// TIA Portal project "SW-Ixxx-xxxx-01" (V15.1)
// Pruebas

(* hardware
DEVICE "S7-1200 station_1"  S7-1200 Station
   slot 0: "Rack_0"  S7-1200 Rack  Rack  V1.0
   slot 1: "PLC_1"  CPU 1211C DC/DC/Rly  6ES7 211-1HE40-0XB0  V4.2
DEVICE "HMI_1"  KTP400 Basic PN
   slot 0: "HMI_1"  KTP400 Basic PN  6AV2 123-2DB03-0AX0  15.1.0.0
   slot 1: "HMI_RT_1"  KTP400 Basic PN  6AV2 123-2DB03-0AX0  15.1.0.0
   slot 5: "HMI_1.IE_CP_1"  PROFINET Interface  15.0.1.0
      slot 1: "Interfaz PROFINET_1"  PROFINET Interface
         slot 1: "Port_1"  Port
*)

// ===== PLC "PLC_1"  CPU 1211C DC/DC/Rly =====

VAR_GLOBAL   // PLC tag table "Tabla de variables estándar"
   "Clock_Byte" AT %MB0 : Byte;
   "Clock_10Hz" AT %M0.0 : Bool;
   "Clock_5Hz" AT %M0.1 : Bool;
   "Clock_2.5Hz" AT %M0.2 : Bool;
   "Clock_2Hz" AT %M0.3 : Bool;
   "Clock_1.25Hz" AT %M0.4 : Bool;
   "Clock_1Hz" AT %M0.5 : Bool;
   "Clock_0.625Hz" AT %M0.6 : Bool;
   "Clock_0.5Hz" AT %M0.7 : Bool;
   "System_Byte" AT %MB1 : Byte;
   "FirstScan" AT %M1.0 : Bool;
   "DiagStatusUpdate" AT %M1.1 : Bool;
   "AlwaysTRUE" AT %M1.2 : Bool;
   "AlwaysFALSE" AT %M1.3 : Bool;
   "Siempre0_IT" AT %M2.0 : Bool;
   "Siempre1_IT" AT %M2.1 : Bool;
   "Debug_IT" AT %M2.2 : Bool;
END_VAR

TYPE "UDT_Motores"
   STRUCT
      Local : Bool;
      Remoto : Bool;
      Manual : Bool;
      Automatico : Bool;
      Habilitado : Bool;
      Deshabilitado : Bool;
      Motor_Ready : Bool;
      Marcha : Bool;
      Confirmacion_de_marcha : Bool;
      Parada : Bool;
      Reset_segundero : Bool;
      Reset_horometro : Bool;
      Comm_PLC_VDF : Bool;   // 1 = OK; 0 = Sin comunicación
      ReservaBool_6 : Bool;
      ReservaBool_7 : Bool;
      ReservaBool_8 : Bool;   // 1= con al menos un enclavamiento activo
      Segundero : Real;   // Segundos en funcionamiento
      Horometro : Real;   // Horas en funcionamiento
      Estado : Real;   // 0 = s/Alm, 1 = c/AlmACK, 2 = c/AlmNoACK, 3 = CondicInseg
      Enclavamiento : Array[0..15] of Bool;
      Alarma : Array[0..15] of Bool;
      VDF : "UDT_VDF";
   END_STRUCT;
   // // Alarma[0] : Falla arranque
   // // Alarma[1] : Falla parada
   // // Alarma[2] : Falla interruptor
   // // Alarma[3] : Falla VDF
   // // Enclavamiento[0] : Equipo enclavado
   // // Enclavamiento[2] : Enclavamiento 2
   // // Enclavamiento[1] : Enclavamiento 1
   // // Enclavamiento[3] : Enclavamiento 3
   // // Enclavamiento[4] : Enclavamiento 4
   // // Enclavamiento[5] : Enclavamiento 5
   // // Enclavamiento[6] : Enclavamiento 6
   // // Enclavamiento[7] : Enclavamiento 7
   // // Enclavamiento[8] : Enclavamiento 8
   // // Enclavamiento[9] : Enclavamiento 9
   // // Enclavamiento[10] : Enclavamiento 10
   // // Enclavamiento[11] : Enclavamiento 11
   // // Enclavamiento[12] : Enclavamiento 12
   // // Enclavamiento[13] : Enclavamiento 13
   // // Enclavamiento[14] : Enclavamiento 14
   // // Enclavamiento[15] : Enclavamiento 15
END_TYPE

TYPE "UDT_Valvulas"
   STRUCT
      Local : Bool;
      Remoto : Bool;
      Manual : Bool;
      Automatico : Bool;
      Habilitado : Bool;
      Deshabilitado : Bool;
      Apertura : Bool;
      Confirmacion_de_apertura : Bool;
      Cierre : Bool;
      Reset_segundero : Bool;
      Reset_horometro : Bool;
      Abriendo : Bool;
      Cerrando : Bool;
      ReservaBool_13 : Bool;
      ReservaBool_14 : Bool;
      ReservaBool_15 : Bool;
      Segundero : Real;   // Segundos en funcionamiento
      Horometro : Real;   // Horas en funcionamiento
      Estado : Real;   // 0 = s/Alm, 1 = c/AlmACK, 2 = c/AlmNoACK, 3 = CondicInseg
      Enclavamiento : Array[0..15] of Bool;
      Alarma : Array[0..15] of Bool;
   END_STRUCT;
   // // Alarma[0] : Falla apertura
   // // Alarma[1] : Falla cierre
   // // Enclavamiento[0] : Equipo enclavado
   // // Enclavamiento[1] : Enclavamiento 1
   // // Enclavamiento[2] : Enclavamiento 2
   // // Enclavamiento[3] : Enclavamiento 3
   // // Enclavamiento[4] : Enclavamiento 4
   // // Enclavamiento[5] : Enclavamiento 5
   // // Enclavamiento[6] : Enclavamiento 6
   // // Enclavamiento[7] : Enclavamiento 7
   // // Enclavamiento[8] : Enclavamiento 8
   // // Enclavamiento[9] : Enclavamiento 9
   // // Enclavamiento[10] : Enclavamiento 10
   // // Enclavamiento[11] : Enclavamiento 11
   // // Enclavamiento[12] : Enclavamiento 12
   // // Enclavamiento[13] : Enclavamiento 13
   // // Enclavamiento[14] : Enclavamiento 14
   // // Enclavamiento[15] : Enclavamiento 15
END_TYPE

TYPE "UDT_Instrumentos"
   STRUCT
      Habilitacion_forzado : Bool;
      Forzado : Bool;
      Reconocer_alarmas_HMI : Bool;
      Reset_valor_acumulado_HMI : Bool;
      Reserva_3 : Bool;
      Reserva_4 : Bool;
      Reserva_5 : Bool;
      Reserva_6 : Bool;
      Reserva_7 : Bool;
      Reserva_8 : Bool;
      Reserva_9 : Bool;
      Reserva_10 : Bool;
      Reserva_11 : Bool;
      Reserva_12 : Bool;
      Reserva_13 : Bool;
      Reserva_14 : Bool;
      Valor_medido : Int;
      Valor_normalizado : Real;
      Valor_escalado : Real;
      Valor_escalado_x_seg : Real;
      Valor_acumulado : Real;
      Seteo : Array[0..6] of Real;
      Alarma : Array[0..15] of Bool;
   END_STRUCT;
   // // Alarma[0] : Alarma por Valor HH
   // // Alarma[1] : Alarma por Valor H
   // // Alarma[2] : Alarma por Valor L
   // // Alarma[3] : Alarma por Valor LL
   // // Alarma[4] : Fuera de Rango
   // // Seteo[0] : Valor de Forzado
   // // Seteo[1] : Valor escalado superior
   // // Seteo[2] : Valor escalado inferior
   // // Seteo[3] : Valor Alarma HH
   // // Seteo[4] : Valor Alarma H
   // // Seteo[5] : Valor Alarma L
   // // Seteo[6] : Valor Alarma LL
END_TYPE

TYPE "UDT_Generadores"
   STRUCT
      Local : Bool;
      Remoto : Bool;
      Manual : Bool;
      Automatico : Bool;
      Habilitado : Bool;
      Deshabilitado : Bool;
      Marcha : Bool;   // Comando marcha/arranque GE
      Confirmacion_de_marcha : Bool;   // 1 = En marcha; 0 = Detenido
      Parada : Bool;   // Comando parada/apagado GE
      Rearranque_automatico : Bool;   // ReEnvío automático del comando marcha/arranque GE
      Reset_horometro : Bool;
      Comm_PLC_GE : Bool;   // 1 = OK; 0 = Sin comunicación
      Ready : Bool;
      Listo_para_carga : Bool;
      En_calentamiento : Bool;   // Inicio espera calentamiento GE
      Confirmacion_calentamiento : Bool;   // Calentamiento Generador OK
      Estado_Generador : Int;   // 0 = Apagado; 1 = En arranque; 2 = Listo para Carga; 3 = En Calentamiento
      Cant_arranques_falla : Int;
      Cant_max_rearranques : Int;
      Calentamiento_et_seg : Int;
      Tiempo_apagado_et_Seg : Int;
      Tiempo_calentamiento : Time;
      Segundero : Real;   // Segundos en funcionamiento
      Horometro : Real;   // Horas en funcionamiento
      Estado : Real;   // 0 = s/Alm, 1 = c/AlmACK, 2 = c/AlmNoACK, 3 = CondicInseg
      Enclavamiento : Array[0..15] of Bool;
      Alarma : Array[0..15] of Bool;
   END_STRUCT;
   // // Alarma[0] : Falla al arrancar GE
   // // Alarma[1] : Falla al detenerse GE
   // // Alarma[2] : Alerta de combustible bajo GE
   // // Alarma[3] : Alarma General
   // // Alarma[4] : Falla comunicación con PLC
   // // Enclavamiento[0] : Equipo enclavado
   // // Enclavamiento[1] : Enclavamiento 1
   // // Enclavamiento[2] : Enclavamiento 2
   // // Enclavamiento[3] : Enclavamiento 3
   // // Enclavamiento[4] : Enclavamiento 4
   // // Enclavamiento[5] : Enclavamiento 5
   // // Enclavamiento[6] : Enclavamiento 6
   // // Enclavamiento[7] : Enclavamiento 7
   // // Enclavamiento[8] : Enclavamiento 8
   // // Enclavamiento[9] : Enclavamiento 9
   // // Enclavamiento[10] : Enclavamiento 10
   // // Enclavamiento[11] : Enclavamiento 11
   // // Enclavamiento[12] : Enclavamiento 12
   // // Enclavamiento[13] : Enclavamiento 13
   // // Enclavamiento[14] : Enclavamiento 14
   // // Enclavamiento[15] : Enclavamiento 15
END_TYPE

TYPE "UDT_VDF"
   STRUCT
      Velocidad_RPM_ref : Real;
      Intensidad_ref : Real;
      Tension_ref : Real;
      Potencia_ref : Real;
      Ret_val : Int;
      Telegrama_Control : Array[0..15] of Word;
      Telegrama_Estado : Array[0..15] of Word;
   END_STRUCT;
   // // Telegrama_Control[0] : Palabra de mando 1 (STW1)
   // // Telegrama_Control[1] : Consigna principal de velocidad
   // // Telegrama_Estado[0] : Palabra de estado 1 (ZSW1)
   // // Telegrama_Estado[1] : Intensidad real Valor absoluto filtrado
   // // Telegrama_Estado[2] : Tensión de salida filtrada
   // // Telegrama_Estado[3] : Velocidad real filtrada
   // // Telegrama_Estado[4] : Potencia activa real filtrada
   // // Telegrama_Estado[5] : Temperatura en motor
   // // Telegrama_Estado[6] : Frecuencia de salida
   // // Telegrama_Estado[7] : Intensidad de fase Valor real, Suma U, V, W
   // // Telegrama_Estado[8] : Código de fallo actual (FAULT_CODE)
   // // Telegrama_Estado[9] : CU Entradas digitales Estado
   // // Telegrama_Estado[10] : Palabra de estado 2
   // // Telegrama_Estado[11] : Tensión en circuito intermedio Valor real
END_TYPE

// folder: B_FUNCIONES GENERALES/DBs Funciones Generales

DATA_BLOCK "DB_Entradas"   // DB100
{ S7_Optimized_Access := 'FALSE' }
VERSION : 0.1
BEGIN
END_DATA_BLOCK

DATA_BLOCK "DB_Salidas"   // DB101
{ S7_Optimized_Access := 'FALSE' }
VERSION : 0.1
BEGIN
END_DATA_BLOCK

DATA_BLOCK "DB_Enclavamientos"   // DB110
{ S7_Optimized_Access := 'FALSE' }
VERSION : 0.1
BEGIN
END_DATA_BLOCK

DATA_BLOCK "DB_PIDs"   // DB120
{ S7_Optimized_Access := 'FALSE' }
VERSION : 0.1
BEGIN
END_DATA_BLOCK

// folder: C_MOTORES/DBs Motores

DATA_BLOCK "DB_Bombas"   // DB210
{ S7_Optimized_Access := 'FALSE' }
VERSION : 0.1
   VAR
      Bomba1 : "UDT_Motores";
   END_VAR
BEGIN
END_DATA_BLOCK

DATA_BLOCK "DB_Agitadores"   // DB220
{ S7_Optimized_Access := 'FALSE' }
VERSION : 0.1
   VAR
      Agitador1 : "UDT_Motores";
   END_VAR
BEGIN
END_DATA_BLOCK

DATA_BLOCK "DB_Ventiladores"   // DB230
{ S7_Optimized_Access := 'FALSE' }
VERSION : 0.1
   VAR
      Ventilador1 : "UDT_Motores";
   END_VAR
BEGIN
END_DATA_BLOCK

DATA_BLOCK "DB_Cintas"   // DB240
{ S7_Optimized_Access := 'FALSE' }
VERSION : 0.1
   VAR
      Cinta1 : "UDT_Motores";
   END_VAR
BEGIN
END_DATA_BLOCK

// folder: D_VALVULAS/DBs Válvulas

DATA_BLOCK "DB_Valvulas_Solenoides"   // DB310
{ S7_Optimized_Access := 'FALSE' }
VERSION : 0.1
BEGIN
END_DATA_BLOCK

DATA_BLOCK "BLQ_Valvula_Solenoide_0_DB"   // DB311
{ S7_Optimized_Access := 'FALSE' }
VERSION : 0.1
// stored: InstanceOfName BLQ_Valvula_Solenoide
"BLQ_Valvula_Solenoide"
BEGIN
END_DATA_BLOCK

DATA_BLOCK "DB_Valvulas_de_Control"   // DB320
{ S7_Optimized_Access := 'FALSE' }
VERSION : 0.1
BEGIN
END_DATA_BLOCK

// folder: E_INSTRUMENTOS/DBs Instrumentos

DATA_BLOCK "DB_Caudalimetros"   // DB410
{ S7_Optimized_Access := 'FALSE' }
VERSION : 0.1
   VAR
      FIT1 : "UDT_Instrumentos";
   END_VAR
BEGIN
END_DATA_BLOCK

DATA_BLOCK "BLQ_FIT_0_DB"   // DB411
{ S7_Optimized_Access := 'FALSE' }
VERSION : 0.1
// stored: InstanceOfName BLQ_Inst_Analogico
"BLQ_Inst_Analogico"
BEGIN
END_DATA_BLOCK

DATA_BLOCK "DB_Sensores_Nivel"   // DB420
{ S7_Optimized_Access := 'FALSE' }
VERSION : 0.1
   VAR
      LIT1 : "UDT_Instrumentos";
   END_VAR
BEGIN
END_DATA_BLOCK

DATA_BLOCK "BLQ_LIT_0_DB"   // DB421
{ S7_Optimized_Access := 'FALSE' }
VERSION : 0.1
// stored: InstanceOfName BLQ_Inst_Digital
"BLQ_Inst_Digital"
BEGIN
END_DATA_BLOCK

DATA_BLOCK "DB_Sensores_Presion"   // DB430
{ S7_Optimized_Access := 'FALSE' }
VERSION : 0.1
   VAR
      PIT1 : "UDT_Instrumentos";
   END_VAR
BEGIN
END_DATA_BLOCK

DATA_BLOCK "DB_Sensores_Temperatura"   // DB440
{ S7_Optimized_Access := 'FALSE' }
VERSION : 0.1
   VAR
      TIT1 : "UDT_Instrumentos";
   END_VAR
BEGIN
END_DATA_BLOCK

// folder: Y_PASARELAS/DBs Pasarelas

DATA_BLOCK "DB_Pasarela1"   // DB901
{ S7_Optimized_Access := 'FALSE' }
VERSION : 0.1
BEGIN
END_DATA_BLOCK

DATA_BLOCK "DB_Pasarela2"   // DB902
{ S7_Optimized_Access := 'FALSE' }
VERSION : 0.1
BEGIN
END_DATA_BLOCK

// folder: Z_COMM/DBs Comm

DATA_BLOCK "DB_Comm1"   // DB1001
{ S7_Optimized_Access := 'FALSE' }
VERSION : 0.1
BEGIN
END_DATA_BLOCK

DATA_BLOCK "DB_Comm2"   // DB1002
{ S7_Optimized_Access := 'FALSE' }
VERSION : 0.1
BEGIN
END_DATA_BLOCK

// folder: A_OBs

ORGANIZATION_BLOCK "Main"   // OB1, LAD, ProgramCycle
TITLE = "Main Program Sweep (Cycle)"
{ S7_Optimized_Access := 'TRUE' }
VERSION : 0.1
   VAR_INPUT
      Initial_Call : Bool;   // Initial call of this OB
      Remanence : Bool;   // =True, if remanent data are available
   END_VAR
BEGIN

REGION Network 1: Asignación de Entradas (%I) a DB de Entradas
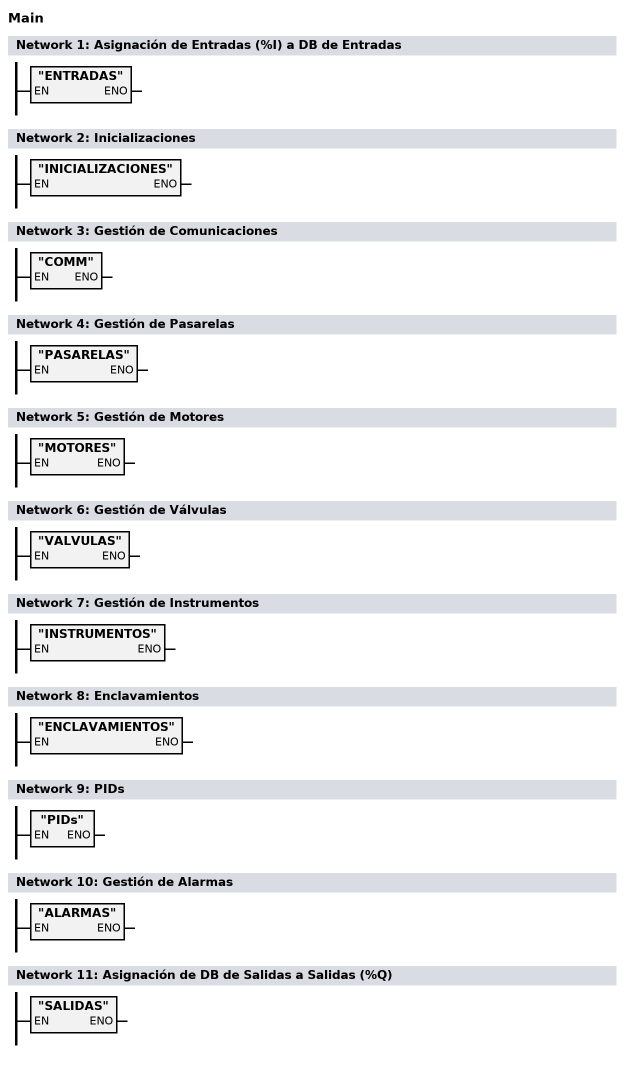
   RUNG wire#powerrail
      "ENTRADAS"()
   END_RUNG
   // the same network as SCL:
   "ENTRADAS"();
END_REGION

REGION Network 2: Inicializaciones
   RUNG wire#powerrail
      "INICIALIZACIONES"()
   END_RUNG
   // the same network as SCL:
   "INICIALIZACIONES"();
END_REGION

REGION Network 3: Gestión de Comunicaciones
   RUNG wire#powerrail
      "COMM"()
   END_RUNG
   // the same network as SCL:
   "COMM"();
END_REGION

REGION Network 4: Gestión de Pasarelas
   RUNG wire#powerrail
      "PASARELAS"()
   END_RUNG
   // the same network as SCL:
   "PASARELAS"();
END_REGION

REGION Network 5: Gestión de Motores
   RUNG wire#powerrail
      "MOTORES"()
   END_RUNG
   // the same network as SCL:
   "MOTORES"();
END_REGION

REGION Network 6: Gestión de Válvulas
   RUNG wire#powerrail
      "VALVULAS"()
   END_RUNG
   // the same network as SCL:
   "VALVULAS"();
END_REGION

REGION Network 7: Gestión de Instrumentos
   RUNG wire#powerrail
      "INSTRUMENTOS"()
   END_RUNG
   // the same network as SCL:
   "INSTRUMENTOS"();
END_REGION

REGION Network 8: Enclavamientos
   RUNG wire#powerrail
      "ENCLAVAMIENTOS"()
   END_RUNG
   // the same network as SCL:
   "ENCLAVAMIENTOS"();
END_REGION

REGION Network 9: PIDs
   RUNG wire#powerrail
      "PIDs"()
   END_RUNG
   // the same network as SCL:
   "PIDs"();
END_REGION

REGION Network 10: Gestión de Alarmas
   RUNG wire#powerrail
      "ALARMAS"()
   END_RUNG
   // the same network as SCL:
   "ALARMAS"();
END_REGION

REGION Network 11: Asignación de DB de Salidas a Salidas (%Q)
   RUNG wire#powerrail
      "SALIDAS"()
   END_RUNG
   // the same network as SCL:
   "SALIDAS"();
END_REGION
END_ORGANIZATION_BLOCK

ORGANIZATION_BLOCK "Startup"   // OB100, LAD, Startup
TITLE = "Complete Restart"
{ S7_Optimized_Access := 'TRUE' }
VERSION : 0.1
   VAR_INPUT
      LostRetentive : Bool;   // True if retentive data are lost
      LostRTC : Bool;   // True if date and time are lost
   END_VAR
BEGIN
END_ORGANIZATION_BLOCK

// folder: B_FUNCIONES GENERALES

FUNCTION "ENTRADAS" : Void   // FC100, LAD
{ S7_Optimized_Access := 'TRUE' }
VERSION : 0.1
// Este bloque es exclusivo para asignar al DB de Entradas TODAS las Entradas físicas (tanto Digitales como Analógicas).
BEGIN
END_FUNCTION

FUNCTION "SALIDAS" : Void   // FC101, LAD
{ S7_Optimized_Access := 'TRUE' }
VERSION : 0.1
// Este bloque es exclusivo para asignar los datos del DB de Salidas a TODAS las Salidas físicas (tanto Digitales como Analógicas).
BEGIN
END_FUNCTION

FUNCTION "INICIALIZACIONES" : Void   // FC102, LAD
{ S7_Optimized_Access := 'TRUE' }
VERSION : 0.1
BEGIN
END_FUNCTION

FUNCTION "ENCLAVAMIENTOS" : Void   // FC110, LAD
{ S7_Optimized_Access := 'TRUE' }
VERSION : 0.1
BEGIN
END_FUNCTION

FUNCTION "PIDs" : Void   // FC120, LAD
TITLE = Selección Local/Remoto y Muestra en HMI quién está operando remotamente al PSJ03
{ S7_Optimized_Access := 'TRUE' }
VERSION : 0.1
BEGIN
END_FUNCTION

// folder: C_MOTORES

FUNCTION "MOTORES" : Void   // FC200, LAD
{ S7_Optimized_Access := 'FALSE' }
VERSION : 0.1
BEGIN
END_FUNCTION

FUNCTION "Bombas" : Void   // FC210, LAD
{ S7_Optimized_Access := 'FALSE' }
VERSION : 0.1
BEGIN
END_FUNCTION

FUNCTION "Agitadores" : Void   // FC220, LAD
{ S7_Optimized_Access := 'TRUE' }
VERSION : 0.1
BEGIN
END_FUNCTION

FUNCTION "Ventiladores" : Void   // FC230, LAD
{ S7_Optimized_Access := 'FALSE' }
VERSION : 0.1
BEGIN
END_FUNCTION

FUNCTION "Cintas" : Void   // FC240, LAD
{ S7_Optimized_Access := 'FALSE' }
VERSION : 0.1
BEGIN
END_FUNCTION

// folder: D_VALVULAS

FUNCTION_BLOCK "BLQ_Valvula_Solenoide"   // FB301, LAD
{ S7_Optimized_Access := 'FALSE' }
VERSION : 0.1
   VAR_INPUT
      SIMU : Bool;
      BEC_RES_in : Bool;   // Enclavamientos Habilitados
      SENC_in : Bool;   // Resumen Motor Enclavado
      SPEM1_in : Bool;   // P.E. de PLC1
      SPEM2_in : Bool;   // P.E. de PLC2
      SAUT_in : Bool;   // SISTEMA en AUTO
      SREM_in : Bool;   // SISTEMA en REMOTO
      FTEN_in : Bool;   // Resumen Falla Tension PLC1
      AACC_CIE_in : Bool;   // Falla Accionamiento Cierre
      AACC_APER_in : Bool;   // Falla Accionamiento Apertura
      SABI_in : Bool;   // Confirmacion V.Abierta
      SCER_in : Bool;   // Confirmacion V.Cerrada
   END_VAR
   VAR_OUTPUT
      SABI_to_OWS : Bool;   // Status V.Abierta a OWS
      SCER_to_OWS : Bool;   // Status V.Cerrada a OWS
      SAUT_to_OWS : Bool;
      SPEM1_to_OWS : Bool;   // 0:Presionada
      SPEM2_to_OWS : Bool;   // 0:Presionada
      CAPE_Q : Bool;   // Comando de Apertura
      CCIE_Q : Bool;   // Comando de Cierre
      SPOS_to_OWS : Real;   // EstadoApert (0=cerrada,1=abierta,2=cerrando,3=abriendo)
      SSTA_to_OWS : Real;   // Estado (Sin Alm=0, ConAlmACK=1, ConAlmNoACK=2)
   END_VAR
   VAR_IN_OUT
      CAPE_OWS1 : Bool;   // Comando Apertura OWS1
      CAPE_HMI : Bool;   // Comando Apertura HMI
      CAPE_OWS2 : Bool;   // Comando Apertura OWS2
      CCIE_HMI : Bool;   // Comando Cierre HMI
      CCIE_OWS1 : Bool;   // Comando Cierre OWS1
      CCIE_OWS2 : Bool;   // Comando Cierre OWS2
      "CAPE_Auto#1_in" : Bool;   // Comando de Partida Automatica OPC#1
      "CAPE_Auto#2_in" : Bool;   // Comando de Partida Automatica OPC#2
      "CCIE_Auto#1_in" : Bool;   // Comando de Detencion Automatica OPC#1
      "CCIE_Auto#2_in" : Bool;   // Comando de Detencion Automatica OPC#2
      CRA1 : Bool;   // Comando Reconocer OWS1
      CRA2 : Bool;   // Comando Reconocer OWS2
      CRAE_SIST : Bool;
      CRAE_HMI_GRAL : Bool;
      CRAE_HMI : Bool;
      SRAE : Bool;
      ACIE_TO_OWS : Bool;   // Falla Cierre OWS
      AAPE_TO_OWS : Bool;   // Falla Apertura OWS
      ASEN_TO_OWS : Bool;   // Falla Sensores OWS
      ATEN_TO_OWS : Bool;   // Falla Tension Comando
   END_VAR
   VAR
      ATEN_disp : Bool;
      AAPER : Bool;   // Falla Apertura
      ACIER : Bool;   // Falla de Cierre deducida
      ARDIN : Bool;
      ASEN_disp : Bool;   // Falla de Sensores
      ASEN_AUX : Bool;   // Auxiliar para flanco
      CAPER_REM : Bool;   // Comando Apertura Remoto Procesado
      CCIER_REM : Bool;   // ComandoCierre Remoto Procesado
      CAPER_HMI : Bool;   // Comando Apertura HMI Procesado
      CCIER_HMI : Bool;   // Comando Cierre HMI Procesado
      CAPER_OUT_int : Bool;
      CCIER_OUT_int : Bool;
      CCIER_OUT_AUX : Bool;
      CAPER_OUT_AUX : Bool;
      SABI_INT : Bool;   // Confirmacion interna V.Abierta
      SCER_INT : Bool;   // Confirmacion interna V.Cerrada
      ACIE_disp : Bool;   // Falla de cierre para alarma IN
      AAPE_disp : Bool;   // Falla de apertura para alarma IN
      CRAE_ACIE : Bool;   // Alarma falla Cierre
      CRAE_ACT : Bool;   // Reconocimiento Aun Activo NC
      APRE_INT : Bool;   // Resumen de Fallas NC
      CRAE_AAPE : Bool;   // Alarma falla Apertura
      CRAE_ASEN : Bool;   // Alarma falla Sensor
      CRAE_ATEN : Bool;
      ACIER_disp : Bool;   // Falla Cierre p/procesar
      AAPER_disp : Bool;   // Falla Apertura p/procesar
      TACK : TON_TIME;
      TMR_ARAC_Loc : TON_TIME;
      TMR_ARAC_Rem : TON_TIME;
   END_VAR
   VAR_TEMP   // added for the SCL form of the ladder/FBD networks
      _w1 : Bool;
   END_VAR
BEGIN

REGION Network 1: Confirmacion Apertura (con Sim)
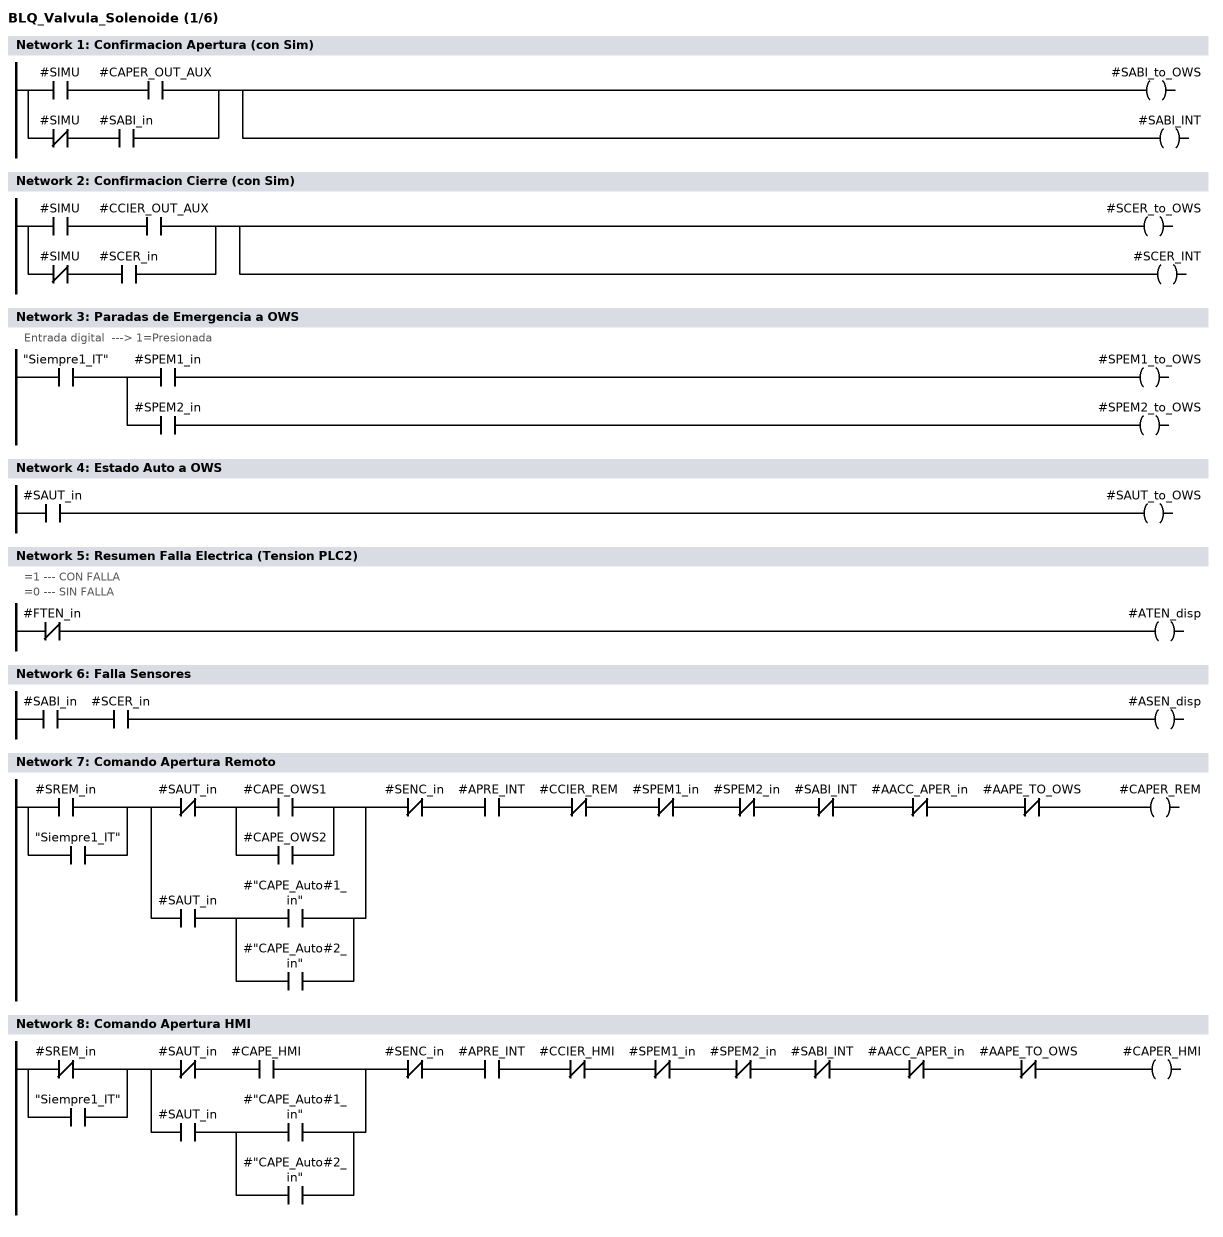
   RUNG wire#powerrail
      Contact( #SIMU )
      Contact( #CAPER_OUT_AUX )
      wire#w1
      Coil( #SABI_to_OWS )
   END_RUNG
   RUNG wire#powerrail
      I_Contact( #SIMU )
      Contact( #SABI_in )
   END_RUNG wire#w1
   RUNG wire#w1
      Coil( #SABI_INT )
   END_RUNG
   // the same network as SCL:
   #SABI_to_OWS := (#SIMU AND #CAPER_OUT_AUX) OR (NOT #SIMU AND #SABI_in);
   #SABI_INT := #SABI_to_OWS;
END_REGION

REGION Network 2: Confirmacion Cierre (con Sim)
   RUNG wire#powerrail
      Contact( #SIMU )
      Contact( #CCIER_OUT_AUX )
      wire#w1
      Coil( #SCER_to_OWS )
   END_RUNG
   RUNG wire#powerrail
      I_Contact( #SIMU )
      Contact( #SCER_in )
   END_RUNG wire#w1
   RUNG wire#w1
      Coil( #SCER_INT )
   END_RUNG
   // the same network as SCL:
   #SCER_to_OWS := (#SIMU AND #CCIER_OUT_AUX) OR (NOT #SIMU AND #SCER_in);
   #SCER_INT := #SCER_to_OWS;
END_REGION

REGION Network 3: Paradas de Emergencia a OWS
   // Entrada digital  ---> 1=Presionada
   RUNG wire#powerrail
      Contact( "Siempre1_IT" )
      wire#w1
      Contact( #SPEM1_in )
      Coil( #SPEM1_to_OWS )
   END_RUNG
   RUNG wire#w1
      Contact( #SPEM2_in )
      Coil( #SPEM2_to_OWS )
   END_RUNG
   // the same network as SCL:
   #SPEM1_to_OWS := "Siempre1_IT" AND #SPEM1_in;
   #SPEM2_to_OWS := "Siempre1_IT" AND #SPEM2_in;
END_REGION

REGION Network 4: Estado Auto a OWS
   RUNG wire#powerrail
      Contact( #SAUT_in )
      Coil( #SAUT_to_OWS )
   END_RUNG
   // the same network as SCL:
   #SAUT_to_OWS := #SAUT_in;
END_REGION

REGION Network 5: Resumen Falla Electrica (Tension PLC2)
   // =1 --- CON FALLA
   // =0 --- SIN FALLA
   RUNG wire#powerrail
      I_Contact( #FTEN_in )
      Coil( #ATEN_disp )
   END_RUNG
   // the same network as SCL:
   #ATEN_disp := NOT #FTEN_in;
END_REGION

REGION Network 6: Falla Sensores
   RUNG wire#powerrail
      Contact( #SABI_in )
      Contact( #SCER_in )
      Coil( #ASEN_disp )
   END_RUNG
   // the same network as SCL:
   #ASEN_disp := #SABI_in AND #SCER_in;
END_REGION

REGION Network 7: Comando Apertura Remoto
   RUNG wire#powerrail
      Contact( #SREM_in )
      wire#w1
      I_Contact( #SAUT_in )
      wire#w2
      Contact( #CAPE_OWS1 )
      wire#w3
      I_Contact( #SENC_in )
      Contact( #APRE_INT )
      I_Contact( #CCIER_REM )
      I_Contact( #SPEM1_in )
      I_Contact( #SPEM2_in )
      I_Contact( #SABI_INT )
      I_Contact( #AACC_APER_in )
      I_Contact( #AAPE_TO_OWS )
      Coil( #CAPER_REM )
   END_RUNG
   RUNG wire#powerrail
      Contact( "Siempre1_IT" )
   END_RUNG wire#w1
   RUNG wire#w2
      Contact( #CAPE_OWS2 )
   END_RUNG wire#w3
   RUNG wire#w1
      Contact( #SAUT_in )
      wire#w4
      Contact( #"CAPE_Auto#1_in" )
   END_RUNG wire#w3
   RUNG wire#w4
      Contact( #"CAPE_Auto#2_in" )
   END_RUNG wire#w3
   // the same network as SCL:
   #CAPER_REM := (#SREM_in OR "Siempre1_IT") AND ((NOT #SAUT_in AND (#CAPE_OWS1 OR #CAPE_OWS2)) OR (#SAUT_in AND (#"CAPE_Auto#1_in" OR #"CAPE_Auto#2_in"))) AND NOT #SENC_in AND #APRE_INT AND NOT #CCIER_REM AND NOT #SPEM1_in AND NOT #SPEM2_in AND NOT #SABI_INT AND NOT #AACC_APER_in AND NOT #AAPE_TO_OWS;
END_REGION

REGION Network 8: Comando Apertura HMI
   RUNG wire#powerrail
      I_Contact( #SREM_in )
      wire#w1
      I_Contact( #SAUT_in )
      Contact( #CAPE_HMI )
      wire#w2
      I_Contact( #SENC_in )
      Contact( #APRE_INT )
      I_Contact( #CCIER_HMI )
      I_Contact( #SPEM1_in )
      I_Contact( #SPEM2_in )
      I_Contact( #SABI_INT )
      I_Contact( #AACC_APER_in )
      I_Contact( #AAPE_TO_OWS )
      Coil( #CAPER_HMI )
   END_RUNG
   RUNG wire#powerrail
      Contact( "Siempre1_IT" )
   END_RUNG wire#w1
   RUNG wire#w1
      Contact( #SAUT_in )
      wire#w3
      Contact( #"CAPE_Auto#1_in" )
   END_RUNG wire#w2
   RUNG wire#w3
      Contact( #"CAPE_Auto#2_in" )
   END_RUNG wire#w2
   // the same network as SCL:
   #CAPER_HMI := (NOT #SREM_in OR "Siempre1_IT") AND ((NOT #SAUT_in AND #CAPE_HMI) OR (#SAUT_in AND (#"CAPE_Auto#1_in" OR #"CAPE_Auto#2_in"))) AND NOT #SENC_in AND #APRE_INT AND NOT #CCIER_HMI AND NOT #SPEM1_in AND NOT #SPEM2_in AND NOT #SABI_INT AND NOT #AACC_APER_in AND NOT #AAPE_TO_OWS;
END_REGION

REGION Network 9: Comando Cierre Remoto
   // APRE_INT lo eliminamos de CCIER dado que si existe falla de apertura/cierre y damos comando de cierre, podrian estar las bombas de Analia en marcha.
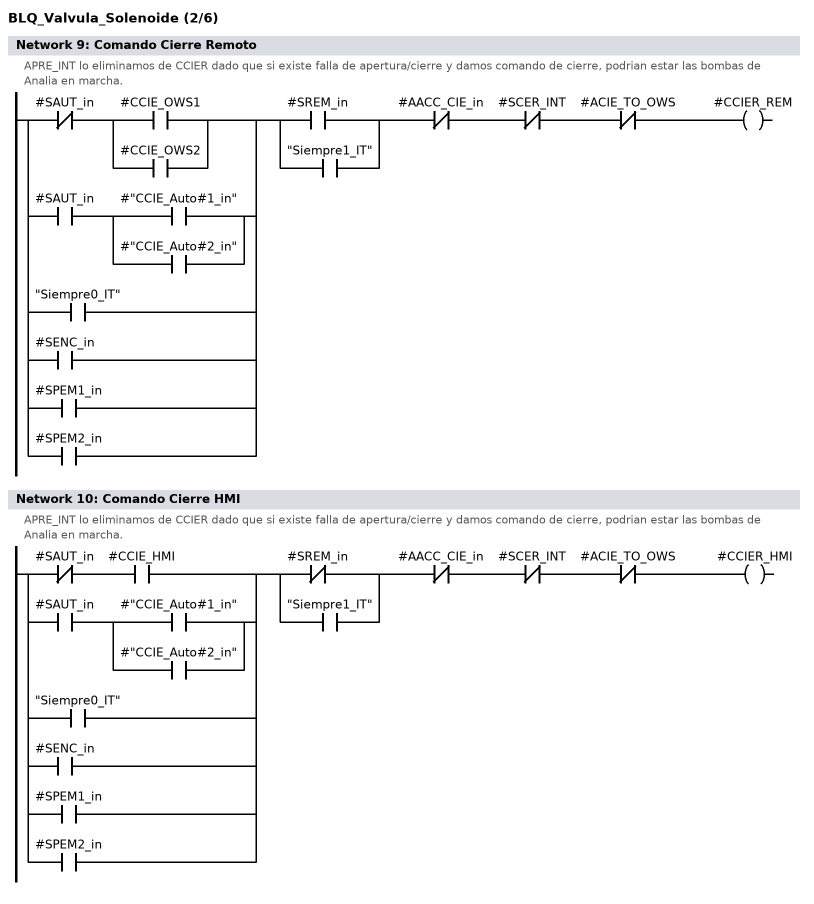
   RUNG wire#powerrail
      I_Contact( #SAUT_in )
      wire#w1
      Contact( #CCIE_OWS1 )
      wire#w2
      Contact( #SREM_in )
      wire#w4
      I_Contact( #AACC_CIE_in )
      I_Contact( #SCER_INT )
      I_Contact( #ACIE_TO_OWS )
      Coil( #CCIER_REM )
   END_RUNG
   RUNG wire#w1
      Contact( #CCIE_OWS2 )
   END_RUNG wire#w2
   RUNG wire#powerrail
      Contact( #SAUT_in )
      wire#w3
      Contact( #"CCIE_Auto#1_in" )
   END_RUNG wire#w2
   RUNG wire#w3
      Contact( #"CCIE_Auto#2_in" )
   END_RUNG wire#w2
   RUNG wire#powerrail
      Contact( "Siempre0_IT" )
   END_RUNG wire#w2
   RUNG wire#powerrail
      Contact( #SENC_in )
   END_RUNG wire#w2
   RUNG wire#powerrail
      Contact( #SPEM1_in )
   END_RUNG wire#w2
   RUNG wire#powerrail
      Contact( #SPEM2_in )
   END_RUNG wire#w2
   RUNG wire#w2
      Contact( "Siempre1_IT" )
   END_RUNG wire#w4
   // the same network as SCL:
   #CCIER_REM := ((NOT #SAUT_in AND (#CCIE_OWS1 OR #CCIE_OWS2)) OR (#SAUT_in AND (#"CCIE_Auto#1_in" OR #"CCIE_Auto#2_in")) OR "Siempre0_IT" OR #SENC_in OR #SPEM1_in OR #SPEM2_in) AND (#SREM_in OR "Siempre1_IT") AND NOT #AACC_CIE_in AND NOT #SCER_INT AND NOT #ACIE_TO_OWS;
END_REGION

REGION Network 10: Comando Cierre HMI
   // APRE_INT lo eliminamos de CCIER dado que si existe falla de apertura/cierre y damos comando de cierre, podrian estar las bombas de Analia en marcha.
   RUNG wire#powerrail
      I_Contact( #SAUT_in )
      Contact( #CCIE_HMI )
      wire#w1
      I_Contact( #SREM_in )
      wire#w3
      I_Contact( #AACC_CIE_in )
      I_Contact( #SCER_INT )
      I_Contact( #ACIE_TO_OWS )
      Coil( #CCIER_HMI )
   END_RUNG
   RUNG wire#powerrail
      Contact( #SAUT_in )
      wire#w2
      Contact( #"CCIE_Auto#1_in" )
   END_RUNG wire#w1
   RUNG wire#w2
      Contact( #"CCIE_Auto#2_in" )
   END_RUNG wire#w1
   RUNG wire#powerrail
      Contact( "Siempre0_IT" )
   END_RUNG wire#w1
   RUNG wire#powerrail
      Contact( #SENC_in )
   END_RUNG wire#w1
   RUNG wire#powerrail
      Contact( #SPEM1_in )
   END_RUNG wire#w1
   RUNG wire#powerrail
      Contact( #SPEM2_in )
   END_RUNG wire#w1
   RUNG wire#w1
      Contact( "Siempre1_IT" )
   END_RUNG wire#w3
   // the same network as SCL:
   #CCIER_HMI := ((NOT #SAUT_in AND #CCIE_HMI) OR (#SAUT_in AND (#"CCIE_Auto#1_in" OR #"CCIE_Auto#2_in")) OR "Siempre0_IT" OR #SENC_in OR #SPEM1_in OR #SPEM2_in) AND (NOT #SREM_in OR "Siempre1_IT") AND NOT #AACC_CIE_in AND NOT #SCER_INT AND NOT #ACIE_TO_OWS;
END_REGION

REGION Network 11: Salida Apertura
   // - Si hay falla de sensores desactivo la salida de Apertura y de Cierre porque nunca va a confirmar ninguna posicion
   // 
   // - Si la valvula confirmo posicion destino desactivo la salida
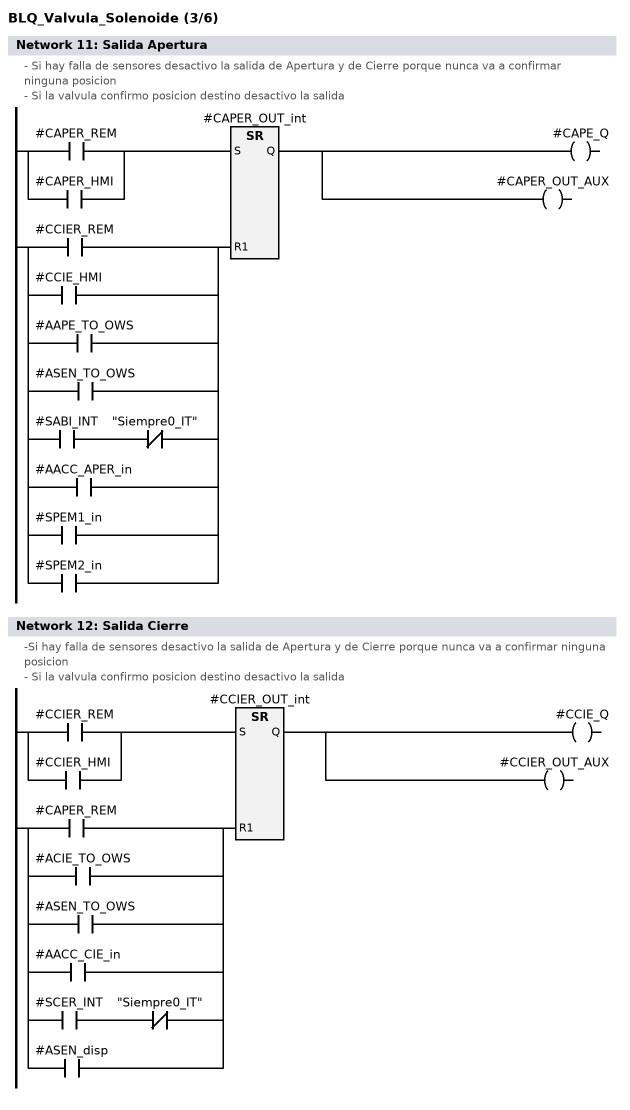
   RUNG wire#powerrail
      Contact( #CAPER_REM )
      wire#w1
      S_SR(operand := #CAPER_OUT_int, r1 := wire#w2)
      wire#w3
      Coil( #CAPE_Q )
   END_RUNG
   RUNG wire#powerrail
      Contact( #CAPER_HMI )
   END_RUNG wire#w1
   RUNG wire#powerrail
      Contact( #CCIER_REM )
   END_RUNG wire#w2
   RUNG wire#powerrail
      Contact( #CCIE_HMI )
   END_RUNG wire#w2
   RUNG wire#powerrail
      Contact( #AAPE_TO_OWS )
   END_RUNG wire#w2
   RUNG wire#powerrail
      Contact( #ASEN_TO_OWS )
   END_RUNG wire#w2
   RUNG wire#powerrail
      Contact( #SABI_INT )
      I_Contact( "Siempre0_IT" )
   END_RUNG wire#w2
   RUNG wire#powerrail
      Contact( #AACC_APER_in )
   END_RUNG wire#w2
   RUNG wire#powerrail
      Contact( #SPEM1_in )
   END_RUNG wire#w2
   RUNG wire#powerrail
      Contact( #SPEM2_in )
   END_RUNG wire#w2
   RUNG wire#w3
      Coil( #CAPER_OUT_AUX )
   END_RUNG
   // the same network as SCL:
   IF #CAPER_REM OR #CAPER_HMI THEN
       #CAPER_OUT_int := TRUE;   // SR flip-flop
   END_IF;
   IF #CCIER_REM OR #CCIE_HMI OR #AAPE_TO_OWS OR #ASEN_TO_OWS OR (#SABI_INT AND NOT "Siempre0_IT") OR #AACC_APER_in OR #SPEM1_in OR #SPEM2_in THEN
       #CAPER_OUT_int := FALSE;
   END_IF;
   #CAPE_Q := #CAPER_OUT_int;
   #CAPER_OUT_AUX := #CAPER_OUT_int;
END_REGION

REGION Network 12: Salida Cierre
   // -Si hay falla de sensores desactivo la salida de Apertura y de Cierre porque nunca va a confirmar ninguna posicion
   // 
   // - Si la valvula confirmo posicion destino desactivo la salida
   RUNG wire#powerrail
      Contact( #CCIER_REM )
      wire#w1
      S_SR(operand := #CCIER_OUT_int, r1 := wire#w2)
      wire#w3
      Coil( #CCIE_Q )
   END_RUNG
   RUNG wire#powerrail
      Contact( #CCIER_HMI )
   END_RUNG wire#w1
   RUNG wire#powerrail
      Contact( #CAPER_REM )
   END_RUNG wire#w2
   RUNG wire#powerrail
      Contact( #ACIE_TO_OWS )
   END_RUNG wire#w2
   RUNG wire#powerrail
      Contact( #ASEN_TO_OWS )
   END_RUNG wire#w2
   RUNG wire#powerrail
      Contact( #AACC_CIE_in )
   END_RUNG wire#w2
   RUNG wire#powerrail
      Contact( #SCER_INT )
      I_Contact( "Siempre0_IT" )
   END_RUNG wire#w2
   RUNG wire#powerrail
      Contact( #ASEN_disp )
   END_RUNG wire#w2
   RUNG wire#w3
      Coil( #CCIER_OUT_AUX )
   END_RUNG
   // the same network as SCL:
   IF #CCIER_REM OR #CCIER_HMI THEN
       #CCIER_OUT_int := TRUE;   // SR flip-flop
   END_IF;
   IF #CAPER_REM OR #ACIE_TO_OWS OR #ASEN_TO_OWS OR #AACC_CIE_in OR (#SCER_INT AND NOT "Siempre0_IT") OR #ASEN_disp THEN
       #CCIER_OUT_int := FALSE;
   END_IF;
   #CCIE_Q := #CCIER_OUT_int;
   #CCIER_OUT_AUX := #CCIER_OUT_int;
END_REGION

REGION Network 13: Estado de Apertura
   // Estados:
   // 0=cerrada
   // 1=abierta
   // 2=cerrando
   // 3=abriendo
   // 4=posicion desconocida
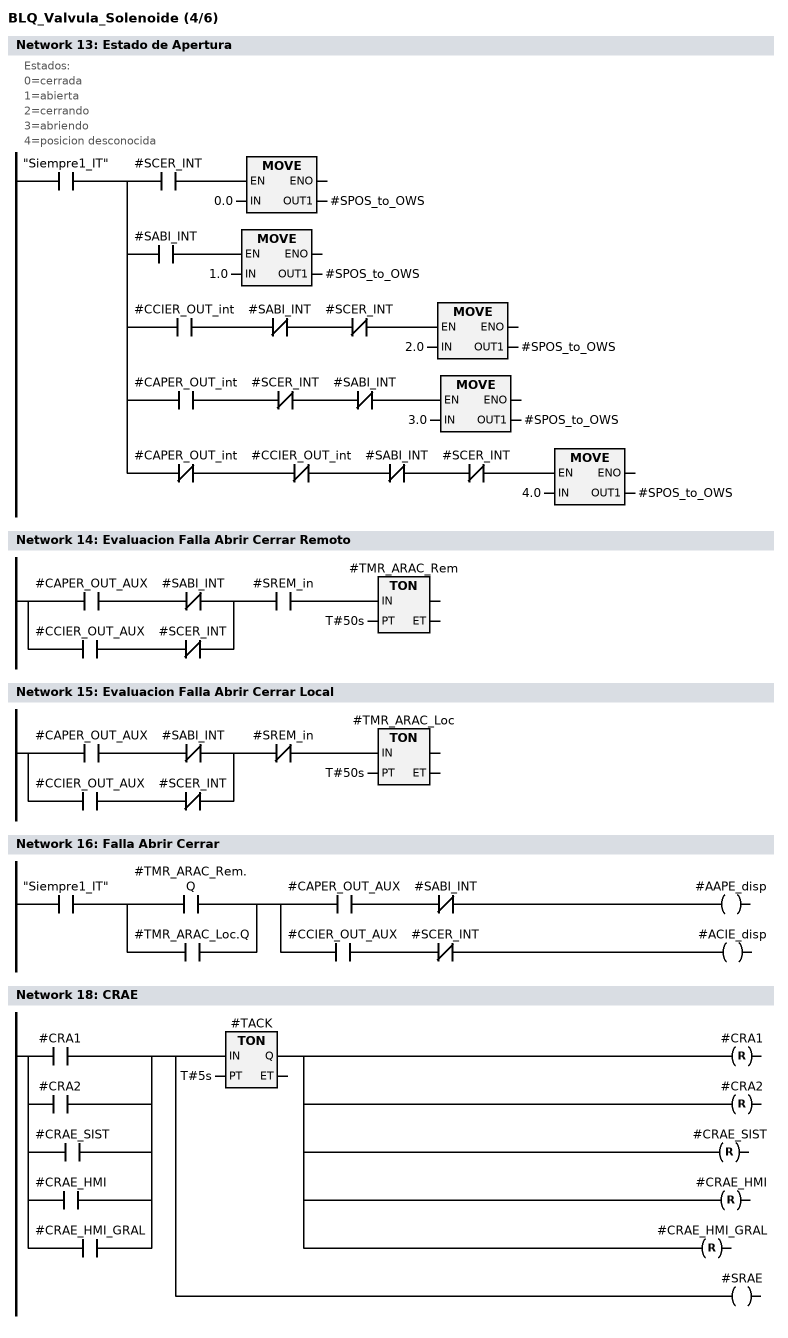
   RUNG wire#powerrail
      Contact( "Siempre1_IT" )
      wire#w1
      Contact( #SCER_INT )
      { S7_GenerateENO := "TRUE" } Move(in := 0.0, out1 => #SPOS_to_OWS)
   END_RUNG
   RUNG wire#w1
      Contact( #SABI_INT )
      { S7_GenerateENO := "TRUE" } Move(in := 1.0, out1 => #SPOS_to_OWS)
   END_RUNG
   RUNG wire#w1
      Contact( #CCIER_OUT_int )
      I_Contact( #SABI_INT )
      I_Contact( #SCER_INT )
      { S7_GenerateENO := "TRUE" } Move(in := 2.0, out1 => #SPOS_to_OWS)
   END_RUNG
   RUNG wire#w1
      Contact( #CAPER_OUT_int )
      I_Contact( #SCER_INT )
      I_Contact( #SABI_INT )
      { S7_GenerateENO := "TRUE" } Move(in := 3.0, out1 => #SPOS_to_OWS)
   END_RUNG
   RUNG wire#w1
      I_Contact( #CAPER_OUT_int )
      I_Contact( #CCIER_OUT_int )
      I_Contact( #SABI_INT )
      I_Contact( #SCER_INT )
      { S7_GenerateENO := "TRUE" } Move(in := 4.0, out1 => #SPOS_to_OWS)
   END_RUNG
   // the same network as SCL:
   IF "Siempre1_IT" AND #SCER_INT THEN #SPOS_to_OWS := 0.0; END_IF;
   IF "Siempre1_IT" AND #SABI_INT THEN #SPOS_to_OWS := 1.0; END_IF;
   IF "Siempre1_IT" AND #CCIER_OUT_int AND NOT #SABI_INT AND NOT #SCER_INT THEN #SPOS_to_OWS := 2.0; END_IF;
   IF "Siempre1_IT" AND #CAPER_OUT_int AND NOT #SCER_INT AND NOT #SABI_INT THEN #SPOS_to_OWS := 3.0; END_IF;
   IF "Siempre1_IT" AND NOT #CAPER_OUT_int AND NOT #CCIER_OUT_int AND NOT #SABI_INT AND NOT #SCER_INT THEN
       #SPOS_to_OWS := 4.0;
   END_IF;
END_REGION

REGION Network 14: Evaluacion Falla Abrir Cerrar Remoto
   #TMR_ARAC_Rem(IN := ((#CAPER_OUT_AUX AND NOT #SABI_INT) OR (#CCIER_OUT_AUX AND NOT #SCER_INT)) AND #SREM_in,   // TON
                 PT := T#50s);
END_REGION

REGION Network 15: Evaluacion Falla Abrir Cerrar Local
   #TMR_ARAC_Loc(IN := ((#CAPER_OUT_AUX AND NOT #SABI_INT) OR (#CCIER_OUT_AUX AND NOT #SCER_INT)) AND NOT #SREM_in,   // TON
                 PT := T#50s);
END_REGION

REGION Network 16: Falla Abrir Cerrar
   RUNG wire#powerrail
      Contact( "Siempre1_IT" )
      wire#w1
      Contact( #TMR_ARAC_Rem.Q )
      wire#w2
      Contact( #CAPER_OUT_AUX )
      I_Contact( #SABI_INT )
      Coil( #AAPE_disp )
   END_RUNG
   RUNG wire#w1
      Contact( #TMR_ARAC_Loc.Q )
   END_RUNG wire#w2
   RUNG wire#w2
      Contact( #CCIER_OUT_AUX )
      I_Contact( #SCER_INT )
      Coil( #ACIE_disp )
   END_RUNG
   // the same network as SCL:
   #_w1 := "Siempre1_IT" AND (#TMR_ARAC_Rem.Q OR #TMR_ARAC_Loc.Q);
   #AAPE_disp := #_w1 AND #CAPER_OUT_AUX AND NOT #SABI_INT;
   #ACIE_disp := #_w1 AND #CCIER_OUT_AUX AND NOT #SCER_INT;
END_REGION

REGION Network 17: ---------- Procesamiento Alarmas ----------------------
END_REGION

REGION Network 18: CRAE
   #_w1 := #CRA1 OR #CRA2 OR #CRAE_SIST OR #CRAE_HMI OR #CRAE_HMI_GRAL;
   #TACK(IN := #_w1, PT := T#5s);   // TON
   IF #TACK.Q THEN
       #CRA1 := FALSE;
       #CRA2 := FALSE;
       #CRAE_SIST := FALSE;
       #CRAE_HMI := FALSE;
       #CRAE_HMI_GRAL := FALSE;
   END_IF;
   #SRAE := #_w1;
END_REGION

REGION Network 19: Reset ACK
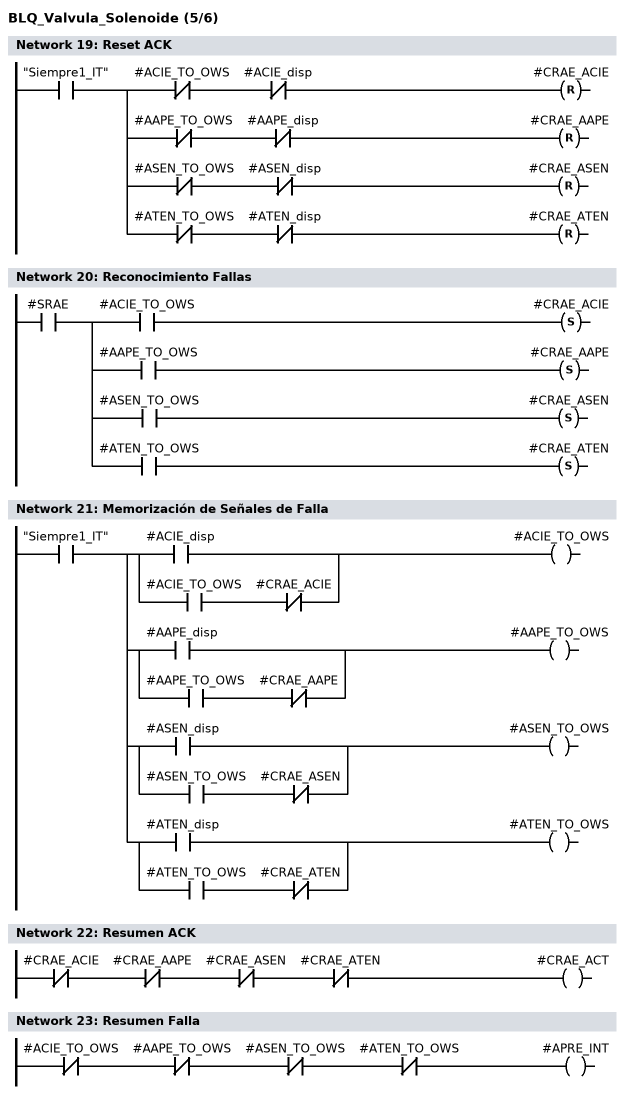
   RUNG wire#powerrail
      Contact( "Siempre1_IT" )
      wire#w1
      I_Contact( #ACIE_TO_OWS )
      I_Contact( #ACIE_disp )
      R_Coil( #CRAE_ACIE )
   END_RUNG
   RUNG wire#w1
      I_Contact( #AAPE_TO_OWS )
      I_Contact( #AAPE_disp )
      R_Coil( #CRAE_AAPE )
   END_RUNG
   RUNG wire#w1
      I_Contact( #ASEN_TO_OWS )
      I_Contact( #ASEN_disp )
      R_Coil( #CRAE_ASEN )
   END_RUNG
   RUNG wire#w1
      I_Contact( #ATEN_TO_OWS )
      I_Contact( #ATEN_disp )
      R_Coil( #CRAE_ATEN )
   END_RUNG
   // the same network as SCL:
   IF "Siempre1_IT" AND NOT #ACIE_TO_OWS AND NOT #ACIE_disp THEN #CRAE_ACIE := FALSE; END_IF;
   IF "Siempre1_IT" AND NOT #AAPE_TO_OWS AND NOT #AAPE_disp THEN #CRAE_AAPE := FALSE; END_IF;
   IF "Siempre1_IT" AND NOT #ASEN_TO_OWS AND NOT #ASEN_disp THEN #CRAE_ASEN := FALSE; END_IF;
   IF "Siempre1_IT" AND NOT #ATEN_TO_OWS AND NOT #ATEN_disp THEN #CRAE_ATEN := FALSE; END_IF;
END_REGION

REGION Network 20: Reconocimiento Fallas
   RUNG wire#powerrail
      Contact( #SRAE )
      wire#w1
      Contact( #ACIE_TO_OWS )
      S_Coil( #CRAE_ACIE )
   END_RUNG
   RUNG wire#w1
      Contact( #AAPE_TO_OWS )
      S_Coil( #CRAE_AAPE )
   END_RUNG
   RUNG wire#w1
      Contact( #ASEN_TO_OWS )
      S_Coil( #CRAE_ASEN )
   END_RUNG
   RUNG wire#w1
      Contact( #ATEN_TO_OWS )
      S_Coil( #CRAE_ATEN )
   END_RUNG
   // the same network as SCL:
   IF #SRAE AND #ACIE_TO_OWS THEN #CRAE_ACIE := TRUE; END_IF;
   IF #SRAE AND #AAPE_TO_OWS THEN #CRAE_AAPE := TRUE; END_IF;
   IF #SRAE AND #ASEN_TO_OWS THEN #CRAE_ASEN := TRUE; END_IF;
   IF #SRAE AND #ATEN_TO_OWS THEN #CRAE_ATEN := TRUE; END_IF;
END_REGION

REGION Network 21: Memorización de Señales de Falla
   RUNG wire#powerrail
      Contact( "Siempre1_IT" )
      wire#w1
      Contact( #ACIE_disp )
      wire#w2
      Coil( #ACIE_TO_OWS )
   END_RUNG
   RUNG wire#w1
      Contact( #ACIE_TO_OWS )
      I_Contact( #CRAE_ACIE )
   END_RUNG wire#w2
   RUNG wire#w1
      Contact( #AAPE_disp )
      wire#w3
      Coil( #AAPE_TO_OWS )
   END_RUNG
   RUNG wire#w1
      Contact( #AAPE_TO_OWS )
      I_Contact( #CRAE_AAPE )
   END_RUNG wire#w3
   RUNG wire#w1
      Contact( #ASEN_disp )
      wire#w4
      Coil( #ASEN_TO_OWS )
   END_RUNG
   RUNG wire#w1
      Contact( #ASEN_TO_OWS )
      I_Contact( #CRAE_ASEN )
   END_RUNG wire#w4
   RUNG wire#w1
      Contact( #ATEN_disp )
      wire#w5
      Coil( #ATEN_TO_OWS )
   END_RUNG
   RUNG wire#w1
      Contact( #ATEN_TO_OWS )
      I_Contact( #CRAE_ATEN )
   END_RUNG wire#w5
   // the same network as SCL:
   #ACIE_TO_OWS := "Siempre1_IT" AND (#ACIE_disp OR (#ACIE_TO_OWS AND NOT #CRAE_ACIE));
   #AAPE_TO_OWS := "Siempre1_IT" AND (#AAPE_disp OR (#AAPE_TO_OWS AND NOT #CRAE_AAPE));
   #ASEN_TO_OWS := "Siempre1_IT" AND (#ASEN_disp OR (#ASEN_TO_OWS AND NOT #CRAE_ASEN));
   #ATEN_TO_OWS := "Siempre1_IT" AND (#ATEN_disp OR (#ATEN_TO_OWS AND NOT #CRAE_ATEN));
END_REGION

REGION Network 22: Resumen ACK
   RUNG wire#powerrail
      I_Contact( #CRAE_ACIE )
      I_Contact( #CRAE_AAPE )
      I_Contact( #CRAE_ASEN )
      I_Contact( #CRAE_ATEN )
      Coil( #CRAE_ACT )
   END_RUNG
   // the same network as SCL:
   #CRAE_ACT := NOT #CRAE_ACIE AND NOT #CRAE_AAPE AND NOT #CRAE_ASEN AND NOT #CRAE_ATEN;
END_REGION

REGION Network 23: Resumen Falla
   RUNG wire#powerrail
      I_Contact( #ACIE_TO_OWS )
      I_Contact( #AAPE_TO_OWS )
      I_Contact( #ASEN_TO_OWS )
      I_Contact( #ATEN_TO_OWS )
      Coil( #APRE_INT )
   END_RUNG
   // the same network as SCL:
   #APRE_INT := NOT #ACIE_TO_OWS AND NOT #AAPE_TO_OWS AND NOT #ASEN_TO_OWS AND NOT #ATEN_TO_OWS;
END_REGION

REGION Network 24: Estado de Alarma
   // Estados:
   // 0-Sin Alarmas
   // 1-Con Alarmas Reconocidas
   // 2-Con Alarmas NO Reconocidas
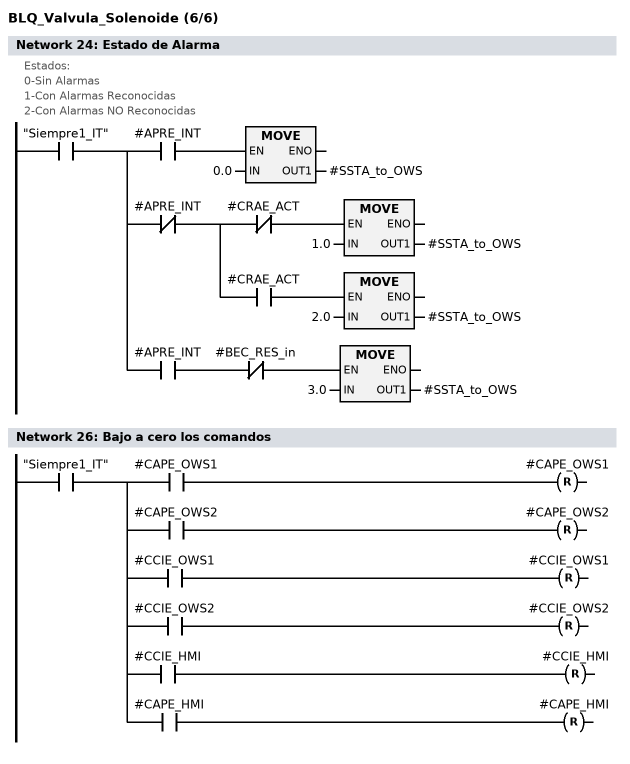
   RUNG wire#powerrail
      Contact( "Siempre1_IT" )
      wire#w1
      Contact( #APRE_INT )
      { S7_GenerateENO := "TRUE" } Move(in := 0.0, out1 => #SSTA_to_OWS)
   END_RUNG
   RUNG wire#w1
      I_Contact( #APRE_INT )
      wire#w2
      I_Contact( #CRAE_ACT )
      { S7_GenerateENO := "TRUE" } Move(in := 1.0, out1 => #SSTA_to_OWS)
   END_RUNG
   RUNG wire#w2
      Contact( #CRAE_ACT )
      { S7_GenerateENO := "TRUE" } Move(in := 2.0, out1 => #SSTA_to_OWS)
   END_RUNG
   RUNG wire#w1
      Contact( #APRE_INT )
      I_Contact( #BEC_RES_in )
      { S7_GenerateENO := "TRUE" } Move(in := 3.0, out1 => #SSTA_to_OWS)
   END_RUNG
   // the same network as SCL:
   IF "Siempre1_IT" AND #APRE_INT THEN #SSTA_to_OWS := 0.0; END_IF;
   #_w1 := "Siempre1_IT" AND NOT #APRE_INT;
   IF #_w1 AND NOT #CRAE_ACT THEN #SSTA_to_OWS := 1.0; END_IF;
   IF #_w1 AND #CRAE_ACT THEN #SSTA_to_OWS := 2.0; END_IF;
   IF "Siempre1_IT" AND #APRE_INT AND NOT #BEC_RES_in THEN #SSTA_to_OWS := 3.0; END_IF;
END_REGION

REGION Network 25: -------------------------------------------------------------------------------------------------------------------------------------------------------
END_REGION

REGION Network 26: Bajo a cero los comandos
   RUNG wire#powerrail
      Contact( "Siempre1_IT" )
      wire#w1
      Contact( #CAPE_OWS1 )
      R_Coil( #CAPE_OWS1 )
   END_RUNG
   RUNG wire#w1
      Contact( #CAPE_OWS2 )
      R_Coil( #CAPE_OWS2 )
   END_RUNG
   RUNG wire#w1
      Contact( #CCIE_OWS1 )
      R_Coil( #CCIE_OWS1 )
   END_RUNG
   RUNG wire#w1
      Contact( #CCIE_OWS2 )
      R_Coil( #CCIE_OWS2 )
   END_RUNG
   RUNG wire#w1
      Contact( #CCIE_HMI )
      R_Coil( #CCIE_HMI )
   END_RUNG
   RUNG wire#w1
      Contact( #CAPE_HMI )
      R_Coil( #CAPE_HMI )
   END_RUNG
   // the same network as SCL:
   IF "Siempre1_IT" AND #CAPE_OWS1 THEN #CAPE_OWS1 := FALSE; END_IF;
   IF "Siempre1_IT" AND #CAPE_OWS2 THEN #CAPE_OWS2 := FALSE; END_IF;
   IF "Siempre1_IT" AND #CCIE_OWS1 THEN #CCIE_OWS1 := FALSE; END_IF;
   IF "Siempre1_IT" AND #CCIE_OWS2 THEN #CCIE_OWS2 := FALSE; END_IF;
   IF "Siempre1_IT" AND #CCIE_HMI THEN #CCIE_HMI := FALSE; END_IF;
   IF "Siempre1_IT" AND #CAPE_HMI THEN #CAPE_HMI := FALSE; END_IF;
END_REGION
END_FUNCTION_BLOCK

FUNCTION "VALVULAS" : Void   // FC300, LAD
{ S7_Optimized_Access := 'TRUE' }
VERSION : 0.1
BEGIN
END_FUNCTION

FUNCTION "Válvulas solenoides" : Void   // FC310, LAD
TITLE = Bloque de gestión de TODAS las válvulas con actuadores solenoides
{ S7_Optimized_Access := 'TRUE' }
VERSION : 0.1
BEGIN

REGION Network 1: "Tag VALVULA" - Descripción
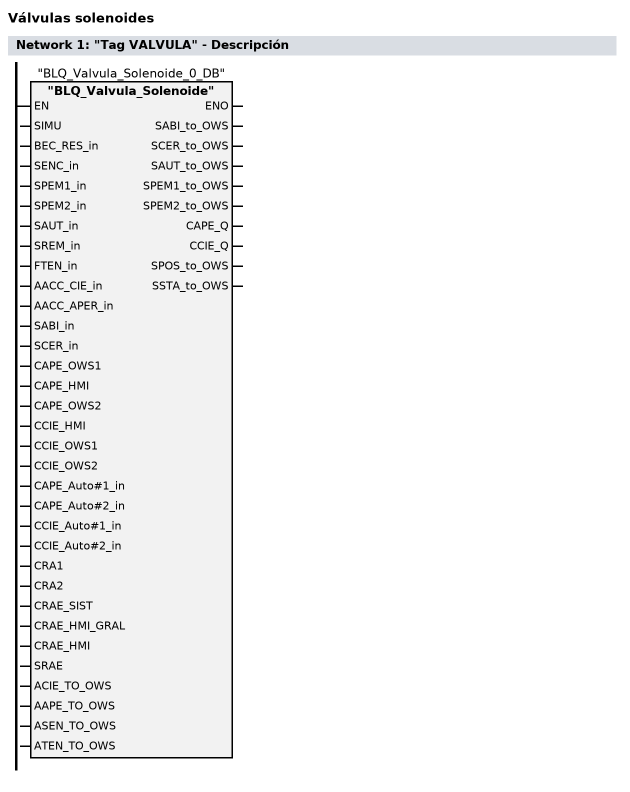
   RUNG wire#powerrail
      "BLQ_Valvula_Solenoide_0_DB"(SIMU :=, BEC_RES_in :=, SENC_in :=, SPEM1_in :=, SPEM2_in :=, SAUT_in :=, SREM_in :=, FTEN_in :=, AACC_CIE_in :=, AACC_APER_in :=, SABI_in :=, SCER_in :=, CAPE_OWS1 :=, CAPE_HMI :=, CAPE_OWS2 :=, CCIE_HMI :=, CCIE_OWS1 :=, CCIE_OWS2 :=, "CAPE_Auto#1_in" :=, "CAPE_Auto#2_in" :=, "CCIE_Auto#1_in" :=, "CCIE_Auto#2_in" :=, CRA1 :=, CRA2 :=, CRAE_SIST :=, CRAE_HMI_GRAL :=, CRAE_HMI :=, SRAE :=, ACIE_TO_OWS :=, AAPE_TO_OWS :=, ASEN_TO_OWS :=, ATEN_TO_OWS :=, SABI_to_OWS =>, SCER_to_OWS =>, SAUT_to_OWS =>, SPEM1_to_OWS =>, SPEM2_to_OWS =>, CAPE_Q =>, CCIE_Q =>, SPOS_to_OWS =>, SSTA_to_OWS =>)
   END_RUNG
   // the same network as SCL:
   "BLQ_Valvula_Solenoide_0_DB"();   // "BLQ_Valvula_Solenoide"
END_REGION
END_FUNCTION

FUNCTION "Válvulas de control" : Void   // FC320, LAD
TITLE = Bloque de gestión de TODAS las válvulas de control
{ S7_Optimized_Access := 'TRUE' }
VERSION : 0.1
BEGIN

REGION Network 1: "Tag CV" - Descripción
END_REGION
END_FUNCTION

// folder: E_INSTRUMENTOS

FUNCTION_BLOCK "BLQ_Inst_Analogico"   // FB401, LAD
TITLE = Bloque de Manejo de Instrumento Analógico
{ S7_Optimized_Access := 'FALSE' }
VERSION : 0.1
   VAR_INPUT
      BHAB : Bool;   // Comando de Habilitación de Forzado desde SCADA
      BBIP_IN : Bool;   // Instrumentos bipolar DB SCADA
      CRAE_ACT : Bool;   // Reconocimiento Aun Activo NC
      APRE_IN : Bool;   // Resumen de Fallas desde FC Alarms NC
      CHHA : Real;   // Valor de Alarma HH (0=deshab.)
      CHAL : Real;   // Valor de Alarma HG (0=deshab.)
      CLAL : Real;   // Valor de Alarma LO (0=deshab.)
      CLLA : Real;   // Valor de Alarma LL (0=deshab.)
      CVAL : Real;   // Valor de Forzado en Unidad Medida
      SVAL_AI : Real;   // Valor Medido Escalado desde AI
      CRAN : Real;   // Valor p/evaluar ARAN
   END_VAR
   VAR_OUTPUT
      AHHL_disp : Bool;   // Alarma por Valor HH a FC Alms
      AHGL_disp : Bool;   // Alarma por Valor HG a FC Alms
      ALOL_disp : Bool;   // Alarma por Valor LO a FC Alms
      ALLL_disp : Bool;   // Alarma por Valor LL a FC Alms
      ARAN_disp : Bool;   // Alarma por Fuera de Rango a FC Alms
      BBIP : Bool;   // Instrumento Bipolar en DB5
      SVAL : Real;   // Valor Medido en Unidad Medida
      SSTA : Real;   // Estado (Sin Alm=0, ConAlmACK=1, ConAlmNoACK=2)
   END_VAR
   VAR
      CERR_AUX : Real;
      SVAL_INT : Real;   // Valor Escalado Actual para uso Interno
   END_VAR
   VAR_TEMP   // added for the SCL form of the ladder/FBD networks
      _w1 : Bool;
   END_VAR
BEGIN

REGION Network 1: Instrumento Bipolar
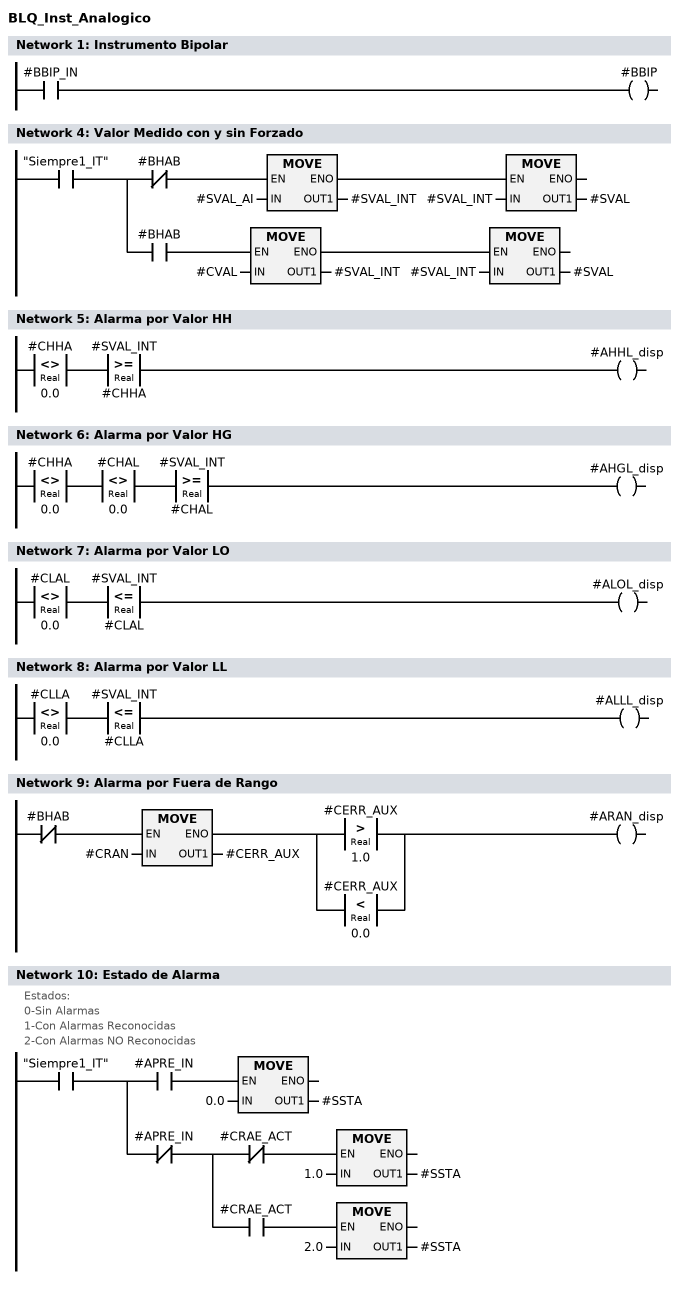
   RUNG wire#powerrail
      Contact( #BBIP_IN )
      Coil( #BBIP )
   END_RUNG
   // the same network as SCL:
   #BBIP := #BBIP_IN;
END_REGION

REGION Network 2: Valor Esc Mín
END_REGION

REGION Network 3: Valor Esc Max
END_REGION

REGION Network 4: Valor Medido con y sin Forzado
   RUNG wire#powerrail
      Contact( "Siempre1_IT" )
      wire#w1
      I_Contact( #BHAB )
      { S7_GenerateENO := "TRUE" } Move(in := #SVAL_AI, out1 => #SVAL_INT)
      { S7_GenerateENO := "TRUE" } Move(in := #SVAL_INT, out1 => #SVAL)
   END_RUNG
   RUNG wire#w1
      Contact( #BHAB )
      { S7_GenerateENO := "TRUE" } Move(in := #CVAL, out1 => #SVAL_INT)
      { S7_GenerateENO := "TRUE" } Move(in := #SVAL_INT, out1 => #SVAL)
   END_RUNG
   // the same network as SCL:
   // ENO of a box is taken as its EN; it also drops when the box reports an error
   IF "Siempre1_IT" AND NOT #BHAB THEN
       #SVAL_INT := #SVAL_AI;
       #SVAL := #SVAL_INT;
   END_IF;
   IF "Siempre1_IT" AND #BHAB THEN
       #SVAL_INT := #CVAL;
       #SVAL := #SVAL_INT;
   END_IF;
END_REGION

REGION Network 5: Alarma por Valor HH
   RUNG wire#powerrail
      { S7_Templates := "SrcType := Real" } NE_Contact(in1 := #CHHA, in2 := 0.0)
      { S7_Templates := "SrcType := Real" } GE_Contact(in1 := #SVAL_INT, in2 := #CHHA)
      Coil( #AHHL_disp )
   END_RUNG
   // the same network as SCL:
   #AHHL_disp := (#CHHA <> 0.0) AND (#SVAL_INT >= #CHHA);
END_REGION

REGION Network 6: Alarma por Valor HG
   RUNG wire#powerrail
      { S7_Templates := "SrcType := Real" } NE_Contact(in1 := #CHHA, in2 := 0.0)
      { S7_Templates := "SrcType := Real" } NE_Contact(in1 := #CHAL, in2 := 0.0)
      { S7_Templates := "SrcType := Real" } GE_Contact(in1 := #SVAL_INT, in2 := #CHAL)
      Coil( #AHGL_disp )
   END_RUNG
   // the same network as SCL:
   #AHGL_disp := (#CHHA <> 0.0) AND (#CHAL <> 0.0) AND (#SVAL_INT >= #CHAL);
END_REGION

REGION Network 7: Alarma por Valor LO
   RUNG wire#powerrail
      { S7_Templates := "SrcType := Real" } NE_Contact(in1 := #CLAL, in2 := 0.0)
      { S7_Templates := "SrcType := Real" } LE_Contact(in1 := #SVAL_INT, in2 := #CLAL)
      Coil( #ALOL_disp )
   END_RUNG
   // the same network as SCL:
   #ALOL_disp := (#CLAL <> 0.0) AND (#SVAL_INT <= #CLAL);
END_REGION

REGION Network 8: Alarma por Valor LL
   RUNG wire#powerrail
      { S7_Templates := "SrcType := Real" } NE_Contact(in1 := #CLLA, in2 := 0.0)
      { S7_Templates := "SrcType := Real" } LE_Contact(in1 := #SVAL_INT, in2 := #CLLA)
      Coil( #ALLL_disp )
   END_RUNG
   // the same network as SCL:
   #ALLL_disp := (#CLLA <> 0.0) AND (#SVAL_INT <= #CLLA);
END_REGION

REGION Network 9: Alarma por Fuera de Rango
   RUNG wire#powerrail
      I_Contact( #BHAB )
      { S7_GenerateENO := "TRUE" } Move(in := #CRAN, out1 => #CERR_AUX)
      wire#w1
      { S7_Templates := "SrcType := Real" } GT_Contact(in1 := #CERR_AUX, in2 := 1.0)
      wire#w2
      Coil( #ARAN_disp )
   END_RUNG
   RUNG wire#w1
      { S7_Templates := "SrcType := Real" } LT_Contact(in1 := #CERR_AUX, in2 := 0.0)
   END_RUNG wire#w2
   // the same network as SCL:
   // ENO of a box is taken as its EN; it also drops when the box reports an error
   IF NOT #BHAB THEN #CERR_AUX := #CRAN; END_IF;
   #ARAN_disp := NOT #BHAB AND ((#CERR_AUX > 1.0) OR (#CERR_AUX < 0.0));
END_REGION

REGION Network 10: Estado de Alarma
   // Estados:
   // 0-Sin Alarmas
   // 1-Con Alarmas Reconocidas
   // 2-Con Alarmas NO Reconocidas
   RUNG wire#powerrail
      Contact( "Siempre1_IT" )
      wire#w1
      Contact( #APRE_IN )
      { S7_GenerateENO := "TRUE" } Move(in := 0.0, out1 => #SSTA)
   END_RUNG
   RUNG wire#w1
      I_Contact( #APRE_IN )
      wire#w2
      I_Contact( #CRAE_ACT )
      { S7_GenerateENO := "TRUE" } Move(in := 1.0, out1 => #SSTA)
   END_RUNG
   RUNG wire#w2
      Contact( #CRAE_ACT )
      { S7_GenerateENO := "TRUE" } Move(in := 2.0, out1 => #SSTA)
   END_RUNG
   // the same network as SCL:
   IF "Siempre1_IT" AND #APRE_IN THEN #SSTA := 0.0; END_IF;
   #_w1 := "Siempre1_IT" AND NOT #APRE_IN;
   IF #_w1 AND NOT #CRAE_ACT THEN #SSTA := 1.0; END_IF;
   IF #_w1 AND #CRAE_ACT THEN #SSTA := 2.0; END_IF;
END_REGION
END_FUNCTION_BLOCK

FUNCTION_BLOCK "BLQ_Inst_Digital"   // FB402, LAD
TITLE = Bloque de Manejo de Switch Digital
{ S7_Optimized_Access := 'FALSE' }
VERSION : 0.1
   VAR_INPUT
      HHFLU_in : Bool;   // Estado detección desde DI
      SVFZ_OWS : Bool;   // Valor de Forzado confirmado
      SHAF_OWS : Bool;   // Confirmacion Comando Habilitación Forzado OWS
      TIPO : Bool;   // Tipo de switch 0=LSL, 1=LSH-LSHH
      CRAE_ACT : Bool;   // Reconocimiento Aun Activo NC
      APRE_in : Bool;   // Resumen de Fallas desde FC Alarms NC
   END_VAR
   VAR_OUTPUT
      ASWH_disp : Bool;   // Disparo Alarma de Switch a FC Alms
      SDET_to_OWS : Bool;   // Estado de Detección
      SSTA_to_OWS : Real;   // Estado (Sin Alm=0, ConAlmACK=1, ConAlmNoACK=2)
      SHAF_to_OWS : Bool;   // Confirmacion Forzado
   END_VAR
   VAR
      SDET_int : Bool;   // Estado de detección uso interno
   END_VAR
   VAR_TEMP   // added for the SCL form of the ladder/FBD networks
      _w1 : Bool;
   END_VAR
BEGIN

REGION Network 1: Valor Detectado con y sin Forzado
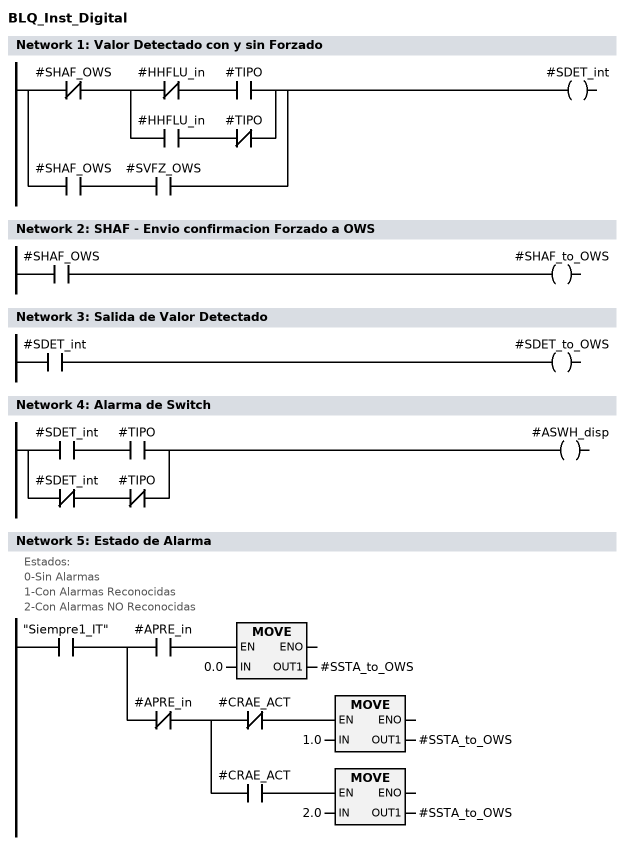
   RUNG wire#powerrail
      I_Contact( #SHAF_OWS )
      wire#w1
      I_Contact( #HHFLU_in )
      Contact( #TIPO )
      wire#w2
      Coil( #SDET_int )
   END_RUNG
   RUNG wire#w1
      Contact( #HHFLU_in )
      I_Contact( #TIPO )
   END_RUNG wire#w2
   RUNG wire#powerrail
      Contact( #SHAF_OWS )
      Contact( #SVFZ_OWS )
   END_RUNG wire#w2
   // the same network as SCL:
   #SDET_int := (NOT #SHAF_OWS AND ((NOT #HHFLU_in AND #TIPO) OR (#HHFLU_in AND NOT #TIPO))) OR (#SHAF_OWS AND #SVFZ_OWS);
END_REGION

REGION Network 2: SHAF - Envio confirmacion Forzado a OWS
   RUNG wire#powerrail
      Contact( #SHAF_OWS )
      Coil( #SHAF_to_OWS )
   END_RUNG
   // the same network as SCL:
   #SHAF_to_OWS := #SHAF_OWS;
END_REGION

REGION Network 3: Salida de Valor Detectado
   RUNG wire#powerrail
      Contact( #SDET_int )
      Coil( #SDET_to_OWS )
   END_RUNG
   // the same network as SCL:
   #SDET_to_OWS := #SDET_int;
END_REGION

REGION Network 4: Alarma de Switch
   RUNG wire#powerrail
      Contact( #SDET_int )
      Contact( #TIPO )
      wire#w1
      Coil( #ASWH_disp )
   END_RUNG
   RUNG wire#powerrail
      I_Contact( #SDET_int )
      I_Contact( #TIPO )
   END_RUNG wire#w1
   // the same network as SCL:
   #ASWH_disp := (#SDET_int AND #TIPO) OR (NOT #SDET_int AND NOT #TIPO);
END_REGION

REGION Network 5: Estado de Alarma
   // Estados:
   // 0-Sin Alarmas
   // 1-Con Alarmas Reconocidas
   // 2-Con Alarmas NO Reconocidas
   RUNG wire#powerrail
      Contact( "Siempre1_IT" )
      wire#w1
      Contact( #APRE_in )
      { S7_GenerateENO := "TRUE" } Move(in := 0.0, out1 => #SSTA_to_OWS)
   END_RUNG
   RUNG wire#w1
      I_Contact( #APRE_in )
      wire#w2
      I_Contact( #CRAE_ACT )
      { S7_GenerateENO := "TRUE" } Move(in := 1.0, out1 => #SSTA_to_OWS)
   END_RUNG
   RUNG wire#w2
      Contact( #CRAE_ACT )
      { S7_GenerateENO := "TRUE" } Move(in := 2.0, out1 => #SSTA_to_OWS)
   END_RUNG
   // the same network as SCL:
   IF "Siempre1_IT" AND #APRE_in THEN #SSTA_to_OWS := 0.0; END_IF;
   #_w1 := "Siempre1_IT" AND NOT #APRE_in;
   IF #_w1 AND NOT #CRAE_ACT THEN #SSTA_to_OWS := 1.0; END_IF;
   IF #_w1 AND #CRAE_ACT THEN #SSTA_to_OWS := 2.0; END_IF;
END_REGION
END_FUNCTION_BLOCK

FUNCTION "INSTRUMENTOS" : Void   // FC400, LAD
{ S7_Optimized_Access := 'TRUE' }
VERSION : 0.1
BEGIN
END_FUNCTION

FUNCTION "Caudalímetros" : Void   // FC410, LAD
TITLE = Bloque de gestión de TODOS los FITs
{ S7_Optimized_Access := 'TRUE' }
VERSION : 0.1
BEGIN

REGION Network 1: "Tag FIT" - Descripción
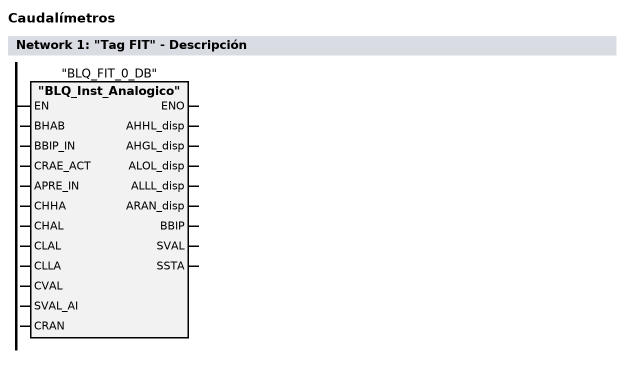
   RUNG wire#powerrail
      "BLQ_FIT_0_DB"(BHAB :=, BBIP_IN :=, CRAE_ACT :=, APRE_IN :=, CHHA :=, CHAL :=, CLAL :=, CLLA :=, CVAL :=, SVAL_AI :=, CRAN :=, AHHL_disp =>, AHGL_disp =>, ALOL_disp =>, ALLL_disp =>, ARAN_disp =>, BBIP =>, SVAL =>, SSTA =>)
   END_RUNG
   // the same network as SCL:
   "BLQ_FIT_0_DB"();   // "BLQ_Inst_Analogico"
END_REGION
END_FUNCTION

FUNCTION "Sensores de Nivel" : Void   // FC420, LAD
TITLE = Bloque de gestión de TODOS los LITs
{ S7_Optimized_Access := 'TRUE' }
VERSION : 0.1
BEGIN

REGION Network 1: "Tag LIT" - Descripción
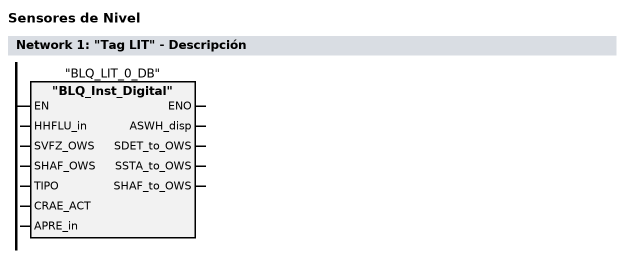
   RUNG wire#powerrail
      "BLQ_LIT_0_DB"(HHFLU_in :=, SVFZ_OWS :=, SHAF_OWS :=, TIPO :=, CRAE_ACT :=, APRE_in :=, ASWH_disp =>, SDET_to_OWS =>, SSTA_to_OWS =>, SHAF_to_OWS =>)
   END_RUNG
   // the same network as SCL:
   "BLQ_LIT_0_DB"();   // "BLQ_Inst_Digital"
END_REGION
END_FUNCTION

FUNCTION "Sensores de Presión" : Void   // FC430, LAD
{ S7_Optimized_Access := 'TRUE' }
VERSION : 0.1
BEGIN
END_FUNCTION

FUNCTION "Sensores de Temperatura" : Void   // FC440, LAD
{ S7_Optimized_Access := 'TRUE' }
VERSION : 0.1
BEGIN
END_FUNCTION

// folder: X_ALARMAS

FUNCTION "ALARMAS" : Void   // FC800, LAD
{ S7_Optimized_Access := 'TRUE' }
VERSION : 0.1
BEGIN
END_FUNCTION

// folder: Y_PASARELAS

FUNCTION "PASARELAS" : Void   // FC900, LAD
{ S7_Optimized_Access := 'TRUE' }
VERSION : 0.1
BEGIN
END_FUNCTION

FUNCTION "Pasarela1" : Void   // FC901, LAD
{ S7_Optimized_Access := 'TRUE' }
VERSION : 0.1
BEGIN
END_FUNCTION

FUNCTION "Pasarela2" : Void   // FC902, LAD
{ S7_Optimized_Access := 'TRUE' }
VERSION : 0.1
BEGIN
END_FUNCTION

// folder: Z_COMM

FUNCTION "COMM" : Void   // FC1000, LAD
{ S7_Optimized_Access := 'FALSE' }
VERSION : 0.1
BEGIN
END_FUNCTION

FUNCTION "Comm1" : Void   // FC1001, LAD
{ S7_Optimized_Access := 'FALSE' }
VERSION : 0.1
BEGIN
END_FUNCTION

FUNCTION "Comm2" : Void   // FC1002, LAD
{ S7_Optimized_Access := 'FALSE' }
VERSION : 0.1
BEGIN
END_FUNCTION

(* ===== HMI "HMI_RT_1" =====
system functions are stored by id; their names below are inferred from use
connection "HMI_Conexión_1": ETHERNET, SMART_S7_1200_OMS

Template "Plantilla_1" 480x272
   Button "Salir" at 388,227 size 63x44; TextOff 'Salir'; PictureOff "ExitRuntime_KTP400_Basic_PN_TR"; PictureOn "ExitRuntime_KTP400_Basic_PN_TR"
      on Release: StopRuntime(0)
   Button "Iniciar sesión" at 268,227 size 63x44; TextOff 'Iniciar sesión'; PictureOff "Login_KTP400_Basic_PN_TR"; PictureOn "Login_KTP400_Basic_PN_TR"
      on Release: function_a2a04561()
   Button "Avisos" at 148,227 size 63x44; TextOff 'Avisos'; PictureOff "AlarmDisplay_KTP400_Basic_PN_TR"; PictureOn "AlarmDisplay_KTP400_Basic_PN_TR"
      on Release: function_ef3f5d25("Ventana de avisos_no_acusado", -1)
   Button "Imagen inicial" at 28,227 size 63x44; TextOff 'Imagen inicial'; PictureOff "NavigateHome_KTP400_Basic_PN_TR"; PictureOn "NavigateHome_KTP400_Basic_PN_TR"
      on Release: ActivateScreen("Imagen raíz", 0)

screen "Imagen raíz" 480x272, template "Plantilla_1"
   TextField "HmiScreenItemData" at 48,100 size 384x22; Text 'Bienvenido a HMI_1 (KTP400 Basic+ PN)!'
   Button "Imagen0" at 1,1 size 157x30; TextOff 'Imagen0'
      on Release: ActivateScreen("Imagen0", 0)
   Button "Imágenes de sistema" at 1,32 size 157x30; TextOff 'Imágenes de siste...'
      on Release: ActivateScreen("Imágenes de sistema", 0)

screen "Imagen0" 480x272, template "Plantilla_1"
   TextField "HmiScreenItemData" at 48,100 size 384x22; Text 'Imagen0'
   Button "Atrás" at 1,1 size 157x30; TextOff 'Atrás'
      on Release: ActivateScreen("Imagen raíz", 0)

screen "Imágenes de sistema" 480x272, template "Plantilla_1"
   TextField "HmiScreenItemData" at 48,100 size 384x22; Text 'Imágenes de sistema'
   Button "Atrás" at 1,1 size 157x30; TextOff 'Atrás'
      on Release: ActivateScreen("Imagen raíz", 0)
   Button "Diagnóstico de sistema SIMATIC PLC" at 1,32 size 157x30; TextOff 'Diagnóstico de sist...'
      on Release: ActivateScreen("Diagnóstico de sistema SIMATIC PLC", 0)
   Button "Información del proyecto" at 1,63 size 157x30; TextOff 'Información del pr...'
      on Release: ActivateScreen("Información del proyecto", 0)
   Button "Administración de usuarios" at 1,94 size 157x30; TextOff 'Administración de u...'
      on Release: ActivateScreen("Administración de usuarios", 0)
   Button "Información de sistema" at 1,125 size 157x30; TextOff 'Información de sist...'
      on Release: ActivateScreen("Información de sistema", 0)
   Button "Tareas varias" at 1,156 size 157x30; TextOff 'Tareas varias'
      on Release: ActivateScreen("Tareas varias", 0)

screen "Diagnóstico de sistema SIMATIC PLC" 480x272, template "Plantilla_1"
   SysDiagControl "HmiScreenItemData" at 1,32 size 476x188
   Button "Atrás" at 1,1 size 157x30; TextOff 'Atrás'
      on Release: ActivateScreen("Imágenes de sistema", 0)

screen "Información del proyecto" 480x272, template "Plantilla_1"
   TextField "HmiScreenItemData" at 4,33 size 184x20; Text 'Nombre del proyecto:'
   TextField "HmiScreenItemData_1" at 192,33 size 284x20; Text 'Proyecto1'
   TextField "HmiScreenItemData_2" at 4,54 size 184x20; Text 'Creado:'
   TextField "HmiScreenItemData_3" at 192,54 size 284x20; Text '15/03/2022 11:15:20'
   TextField "HmiScreenItemData_4" at 4,75 size 184x20; Text 'Autor:'
   TextField "HmiScreenItemData_5" at 192,75 size 284x20; Text 'Emilio Ryan'
   TextField "HmiScreenItemData_6" at 4,96 size 184x20; Text 'Descripción:'
   TextField "HmiScreenItemData_7" at 192,96 size 284x20; Text 'Pruebas'
   Button "Atrás" at 1,1 size 157x30; TextOff 'Atrás'
      on Release: ActivateScreen("Imágenes de sistema", 0)

screen "Administración de usuarios" 480x272, template "Plantilla_1"
   UserView "HmiScreenItemData" at 1,32 size 476x188
   Button "Atrás" at 1,1 size 157x30; TextOff 'Atrás'
      on Release: ActivateScreen("Imágenes de sistema", 0)

screen "Información de sistema" 480x272, template "Plantilla_1"
   TextField "HmiScreenItemData" at 4,33 size 184x20; Text 'Tipo de panel:'
   TextField "HmiScreenItemData_1" at 192,33 size 284x20; Text 'KTP400 Basic+ PN 15.1.0.0'
   TextField "HmiScreenItemData_2" at 4,54 size 184x20; Text 'Conexión:'
   TextField "HmiScreenItemData_3" at 192,54 size 284x20; Text 'PROFINET (X1)'
   TextField "HmiScreenItemData_4" at 4,75 size 184x20; Text 'Controlador:'
   TextField "HmiScreenItemData_5" at 192,75 size 284x20; Text 'SIMATIC S7 1200'
   Button "Atrás" at 1,1 size 157x30; TextOff 'Atrás'
      on Release: ActivateScreen("Imágenes de sistema", 0)

screen "Tareas varias" 480x272, template "Plantilla_1"
   Button "Online" at 1,32 size 157x30; TextOff 'Online'
      on Release: function_bb44b551(0)
   Button "Offline" at 1,63 size 157x30; TextOff 'Offline'
      on Release: function_bb44b551(1)
   Button "Transferencia" at 1,94 size 157x30; TextOff 'Transferencia'
      on Release: function_bb44b551(2)
   Button "Cambiar idioma" at 1,125 size 157x30; TextOff 'Cambiar idioma'
      on Release: function_fb9197e8(-1)
   Button "Salir de runtime" at 1,156 size 157x30; TextOff 'Salir de runtime'
      on Release: StopRuntime(0)
   Button "Atrás" at 1,1 size 157x30; TextOff 'Atrás'
      on Release: ActivateScreen("Imágenes de sistema", 0)
*)